KUKA KRL program: MyProgram_316().src

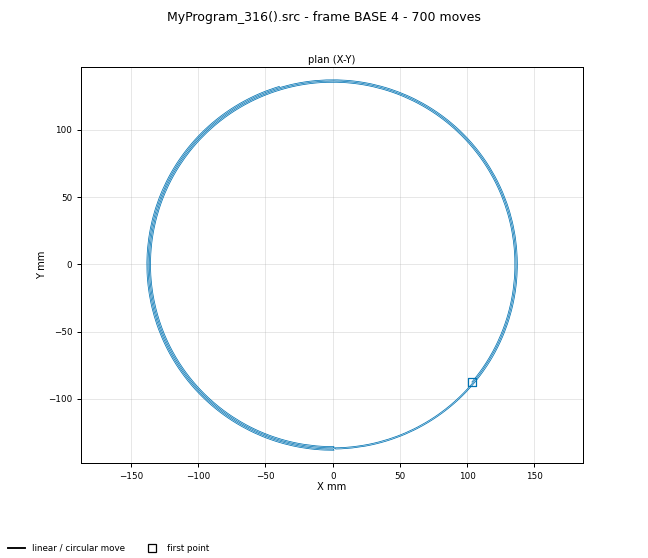
[picture p0: tool path of MyProgram_316().src in frame BASE 4, 700 of 700 moves have a stored position in this frame; points joined in program order, loops and branches not executed]
&ACCESS RVP
&REL 1
&PARAM TEMPLATE = C:\KRC\Roboter\Template\vorgabe
&PARAM EDITMASK = *
DEF MyProgram_316()
; ---- Setting reference (Base) ----
$BASE = BASE_DATA[4]

; --------------------------
; ---- Setting tool (TCP) ----
$TOOL = TOOL_DATA[3]
; --------------------------

$VEL.CP = VEL_APROX_PRINT
Startdeposition()
$VEL.CP = VEL_PRINT
LIN {X 103.5181,Y -87.4443,Z 184,A -35.435,B 3.7699,C 0.2794,E1 3.9046,E2 488.1643} C_DIS
LIN {X 106.5968,Y -83.6627,Z 184,A -33.5084,B 3.7701,C 0.2762,E1 3.9079,E2 486.2534} C_DIS
LIN {X 109.2391,Y -80.182,Z 184,A -31.7632,B 3.7704,C 0.2731,E1 3.9108,E2 484.52} C_DIS
LIN {X 111.321,Y -77.2656,Z 184,A -29.7761,B 3.771,C 0.2642,E1 3.9141,E2 482.4703} C_DIS
LIN {X 113.9076,Y -73.3999,Z 184,A -28.2787,B 3.771,C 0.2647,E1 3.9163,E2 481.0323} C_DIS
LIN {X 116.3066,Y -69.5351,Z 184,A -26.5939,B 3.7711,C 0.2627,E1 3.9187,E2 479.3768} C_DIS
LIN {X 119.2726,Y -64.315,Z 184,A -23.9196,B 3.7716,C 0.2548,E1 3.9223,E2 476.683} C_DIS
LIN {X 121.3738,Y -60.2518,Z 184,A -22.1723,B 3.7718,C 0.2519,E1 3.9245,E2 474.9581} C_DIS
LIN {X 122.8506,Y -57.1807,Z 184,A -20.8286,B 3.772,C 0.2493,E1 3.9261,E2 473.6257} C_DIS
LIN {X 124.2779,Y -54.0078,Z 184,A -19.6123,B 3.772,C 0.2483,E1 3.9274,E2 472.4408} C_DIS
LIN {X 125.1592,Y -51.9333,Z 184,A -18.3421,B 3.7725,C 0.2422,E1 3.9288,E2 471.1292} C_DIS
LIN {X 126.782,Y -47.8354,Z 184,A -16.8653,B 3.7725,C 0.2417,E1 3.9303,E2 469.7006} C_DIS
LIN {X 128.1212,Y -44.1231,Z 184,A -14.9406,B 3.773,C 0.2343,E1 3.9321,E2 467.7417} C_DIS
LIN {X 129.4777,Y -39.9682,Z 184,A -13.2527,B 3.7732,C 0.2311,E1 3.9335,E2 466.0729} C_DIS
LIN {X 130.4392,Y -36.7082,Z 184,A -11.883,B 3.7734,C 0.2279,E1 3.9346,E2 464.7107} C_DIS
LIN {X 131.3258,Y -33.3972,Z 184,A -10.4346,B 3.7736,C 0.2239,E1 3.9356,E2 463.2613} C_DIS
LIN {X 132.2992,Y -29.3141,Z 184,A -8.6511,B 3.7739,C 0.2189,E1 3.9367,E2 461.4754} C_DIS
LIN {X 133.0621,Y -25.6197,Z 184,A -7.2855,B 3.7739,C 0.2171,E1 3.9374,E2 460.1378} C_DIS
LIN {X 133.6399,Y -22.4114,Z 184,A -5.8945,B 3.7742,C 0.2131,E1 3.9381,E2 458.7442} C_DIS
LIN {X 134.2034,Y -18.7486,Z 184,A -4.3975,B 3.7744,C 0.2095,E1 3.9387,E2 457.2549} C_DIS
LIN {X 135.083,Y -10.7221,Z 184,A -1.0365,B 3.7749,C 0.2006,E1 3.9397,E2 453.8983} C_DIS
LIN {X 135.3222,Y -7.0634,Z 184,A 0.376,B 3.7751,C 0.1977,E1 3.9399,E2 452.5023} C_DIS
LIN {X 135.4633,Y -3.4258,Z 184,A 2.0383,B 3.7754,C 0.192,E1 3.94,E2 450.8232} C_DIS
LIN {X 135.4418,Y 4.2013,Z 184,A 5.0751,B 3.7757,C 0.185,E1 3.94,E2 447.8082} C_DIS
LIN {X 135.3131,Y 7.2441,Z 184,A 6.7756,B 3.7761,C 0.1767,E1 3.9397,E2 446.0544} C_DIS
LIN {X 134.9595,Y 12.1833,Z 184,A 8.2582,B 3.7761,C 0.1778,E1 3.9393,E2 444.6481} C_DIS
LIN {X 134.3821,Y 17.4175,Z 184,A 10.3473,B 3.7763,C 0.1731,E1 3.9386,E2 442.5749} C_DIS
LIN {X 133.9505,Y 20.4746,Z 184,A 11.6618,B 3.7764,C 0.1693,E1 3.9381,E2 441.2585} C_DIS
LIN {X 133.4035,Y 23.778,Z 184,A 12.9257,B 3.7765,C 0.1671,E1 3.9375,E2 440.0129} C_DIS
LIN {X 132.7476,Y 27.2026,Z 184,A 14.4382,B 3.7767,C 0.1626,E1 3.9367,E2 438.4947} C_DIS
LIN {X 131.8443,Y 31.2913,Z 184,A 16.18,B 3.7769,C 0.158,E1 3.9356,E2 436.7555} C_DIS
LIN {X 130.9715,Y 34.7611,Z 184,A 17.5774,B 3.777,C 0.1552,E1 3.9346,E2 435.3717} C_DIS
LIN {X 130.0827,Y 37.9517,Z 184,A 18.9487,B 3.7772,C 0.1517,E1 3.9336,E2 434.0034} C_DIS
LIN {X 129.068,Y 41.2706,Z 184,A 20.3738,B 3.7773,C 0.1482,E1 3.9324,E2 432.5828} C_DIS
LIN {X 128.1625,Y 44.0039,Z 184,A 21.9177,B 3.7776,C 0.1413,E1 3.931,E2 430.9974} C_DIS
LIN {X 126.8571,Y 47.635,Z 184,A 23.0833,B 3.7776,C 0.1422,E1 3.9299,E2 429.8894} C_DIS
LIN {X 125.7062,Y 50.594,Z 184,A 24.4415,B 3.7776,C 0.1384,E1 3.9285,E2 428.5286} C_DIS
LIN {X 124.1044,Y 54.4093,Z 184,A 26.2365,B 3.7779,C 0.1334,E1 3.9265,E2 426.7272} C_DIS
LIN {X 122.8136,Y 57.2608,Z 184,A 27.4747,B 3.7779,C 0.1309,E1 3.9251,E2 425.4991} C_DIS
LIN {X 121.1492,Y 60.7072,Z 184,A 29.0707,B 3.7781,C 0.1271,E1 3.9231,E2 423.9053} C_DIS
LIN {X 119.1914,Y 64.4661,Z 184,A 30.7766,B 3.7782,C 0.1235,E1 3.9208,E2 422.2093} C_DIS
LIN {X 116.2038,Y 69.7076,Z 184,A 33.2579,B 3.7784,C 0.118,E1 3.9174,E2 419.7358} C_DIS
LIN {X 113.8832,Y 73.4375,Z 184,A 34.9973,B 3.7784,C 0.1148,E1 3.9148,E2 418.0104} C_DIS
LIN {X 112.1478,Y 76.0606,Z 184,A 36.3024,B 3.7786,C 0.1119,E1 3.9128,E2 416.708} C_DIS
LIN {X 109.5386,Y 79.7729,Z 184,A 38.1589,B 3.7786,C 0.1081,E1 3.9098,E2 414.8587} C_DIS
LIN {X 106.995,Y 83.153,Z 184,A 39.8979,B 3.7788,C 0.1046,E1 3.9068,E2 413.1252} C_DIS
LIN {X 104.2275,Y 86.5968,Z 184,A 41.7072,B 3.7788,C 0.1011,E1 3.9036,E2 411.3227} C_DIS
LIN {X 101.3001,Y 90.004,Z 184,A 43.5795,B 3.779,C 0.0973,E1 3.9002,E2 409.4534} C_DIS
LIN {X 98.7892,Y 92.753,Z 184,A 45.5297,B 3.7792,C 0.09,E1 3.8964,E2 407.4564} C_DIS
LIN {X 95.608,Y 96.0284,Z 184,A 46.8132,B 3.7791,C 0.0928,E1 3.894,E2 406.2524} C_DIS
LIN {X 90.6851,Y 100.691,Z 184,A 49.8084,B 3.7793,C 0.0858,E1 3.8879,E2 403.2412} C_DIS
LIN {X 87.3464,Y 103.6004,Z 184,A 51.6137,B 3.7793,C 0.083,E1 3.884,E2 401.4439} C_DIS
LIN {X 84.0447,Y 106.2967,Z 184,A 53.3461,B 3.7793,C 0.0804,E1 3.8803,E2 399.72} C_DIS
LIN {X 80.6714,Y 108.8786,Z 184,A 55.1005,B 3.7794,C 0.0777,E1 3.8764,E2 397.9706} C_DIS
LIN {X 77.034,Y 111.4822,Z 184,A 56.9839,B 3.7794,C 0.0746,E1 3.8721,E2 396.0881} C_DIS
LIN {X 73.3256,Y 113.9552,Z 184,A 58.8067,B 3.7795,C 0.0722,E1 3.8678,E2 394.2729} C_DIS
LIN {X 69.7051,Y 116.2053,Z 184,A 60.6036,B 3.7795,C 0.0695,E1 3.8635,E2 392.4767} C_DIS
LIN {X 66.7818,Y 117.9097,Z 184,A 61.9456,B 3.7796,C 0.0682,E1 3.8603,E2 391.1456} C_DIS
LIN {X 63.2705,Y 119.8278,Z 184,A 63.5525,B 3.7796,C 0.0667,E1 3.8564,E2 389.549} C_DIS
LIN {X 60.3352,Y 121.3327,Z 184,A 64.9003,B 3.7796,C 0.0652,E1 3.853,E2 388.2071} C_DIS
LIN {X 57.0324,Y 122.9191,Z 184,A 66.4113,B 3.7796,C 0.0636,E1 3.8492,E2 386.7009} C_DIS
LIN {X 54.1496,Y 124.2167,Z 184,A 67.7281,B 3.7797,C 0.0622,E1 3.8459,E2 385.3867} C_DIS
LIN {X 50.7905,Y 125.627,Z 184,A 69.2033,B 3.7797,C 0.061,E1 3.8421,E2 383.9196} C_DIS
LIN {X 47.6823,Y 126.8394,Z 184,A 70.6206,B 3.7797,C 0.0594,E1 3.8384,E2 382.5017} C_DIS
LIN {X 44.4026,Y 128.0243,Z 184,A 72.1122,B 3.7797,C 0.0578,E1 3.8344,E2 381.0083} C_DIS
LIN {X 41.1802,Y 129.0969,Z 184,A 73.6768,B 3.7798,C 0.0552,E1 3.8302,E2 379.4284} C_DIS
LIN {X 37.2623,Y 130.2842,Z 184,A 75.3555,B 3.7798,C 0.0542,E1 3.8258,E2 377.7565} C_DIS
LIN {X 33.5935,Y 131.276,Z 184,A 76.8272,B 3.7798,C 0.0542,E1 3.8218,E2 376.3015} C_DIS
LIN {X 30.4525,Y 132.0401,Z 184,A 78.1762,B 3.7798,C 0.0533,E1 3.8182,E2 374.9551} C_DIS
LIN {X 26.9784,Y 132.7932,Z 184,A 79.7173,B 3.7798,C 0.0519,E1 3.8139,E2 373.4097} C_DIS
LIN {X 22.9319,Y 133.553,Z 184,A 81.4911,B 3.7798,C 0.0506,E1 3.809,E2 371.6326} C_DIS
LIN {X 19.2145,Y 134.1368,Z 184,A 83.0044,B 3.7798,C 0.0505,E1 3.8049,E2 370.1291} C_DIS
LIN {X 15.1542,Y 134.6577,Z 184,A 85.3116,B 3.78,C 0.0449,E1 3.7983,E2 367.7527} C_DIS
LIN {X 10.2568,Y 135.118,Z 184,A 86.7787,B 3.78,C 0.0494,E1 3.7944,E2 366.3607} C_DIS
LIN {X 6.746,Y 135.3382,Z 184,A 88.2689,B 3.78,C 0.049,E1 3.7903,E2 364.8707} C_DIS
LIN {X 2.8347,Y 135.4778,Z 184,A 90.1909,B 3.78,C 0.0465,E1 3.7848,E2 362.9171} C_DIS
LIN {X -4.5052,Y 135.4333,Z 184,A 93.1017,B 3.78,C 0.0479,E1 3.7767,E2 360.0311} C_DIS
LIN {X -8.3822,Y 135.2467,Z 184,A 94.6551,B 3.78,C 0.0487,E1 3.7724,E2 358.489} C_DIS
LIN {X -11.9873,Y 134.9761,Z 184,A 96.6447,B 3.78,C 0.0454,E1 3.7667,E2 356.4445} C_DIS
LIN {X -16.0503,Y 134.5522,Z 184,A 97.9717,B 3.78,C 0.0489,E1 3.7632,E2 355.1668} C_DIS
LIN {X -20.4686,Y 133.9514,Z 184,A 99.7685,B 3.7799,C 0.0501,E1 3.7583,E2 353.3815} C_DIS
LIN {X -23.5464,Y 133.4449,Z 184,A 101.1595,B 3.7799,C 0.0501,E1 3.7544,E2 351.9826} C_DIS
LIN {X -26.9594,Y 132.797,Z 184,A 102.6559,B 3.7799,C 0.0506,E1 3.7503,E2 350.4837} C_DIS
LIN {X -30.9686,Y 131.9221,Z 184,A 104.4857,B 3.7799,C 0.0508,E1 3.7453,E2 348.6435} C_DIS
LIN {X -34.5894,Y 131.0173,Z 184,A 105.9655,B 3.7799,C 0.0525,E1 3.7413,E2 347.1765} C_DIS
LIN {X -37.9806,Y 130.0742,Z 184,A 107.5309,B 3.7799,C 0.053,E1 3.7371,E2 345.6026} C_DIS
LIN {X -42.695,Y 128.6039,Z 184,A 109.5217,B 3.7799,C 0.0553,E1 3.7318,E2 343.6248} C_DIS
LIN {X -45.7334,Y 127.5552,Z 184,A 111.6211,B 3.7799,C 0.0513,E1 3.7261,E2 341.4366} C_DIS
LIN {X -50.6638,Y 125.6781,Z 184,A 113.2742,B 3.7798,C 0.0575,E1 3.722,E2 339.8551} C_DIS
LIN {X -54.6362,Y 124.005,Z 184,A 115.1537,B 3.7798,C 0.059,E1 3.7171,E2 337.97} C_DIS
LIN {X -57.8691,Y 122.5288,Z 184,A 116.6209,B 3.7798,C 0.0609,E1 3.7134,E2 336.508} C_DIS
LIN {X -61.0853,Y 120.9568,Z 184,A 118.6584,B 3.7798,C 0.0592,E1 3.7082,E2 334.4081} C_DIS
LIN {X -65.2213,Y 118.7799,Z 184,A 120.237,B 3.7797,C 0.0644,E1 3.7044,E2 332.8792} C_DIS
LIN {X -69.0275,Y 116.6091,Z 184,A 122.1205,B 3.7797,C 0.0667,E1 3.6999,E2 330.9933} C_DIS
LIN {X -73.0206,Y 114.1504,Z 184,A 124.4662,B 3.7797,C 0.0673,E1 3.6942,E2 328.6049} C_DIS
LIN {X -76.3633,Y 111.9425,Z 184,A 125.8969,B 3.7796,C 0.0715,E1 3.691,E2 327.2075} C_DIS
LIN {X -79.8005,Y 109.5186,Z 184,A 128.3863,B 3.7796,C 0.0699,E1 3.6852,E2 324.6327} C_DIS
LIN {X -84.4566,Y 105.9683,Z 184,A 130.1256,B 3.7794,C 0.0787,E1 3.6816,E2 322.9852} C_DIS
LIN {X -87.6625,Y 103.3326,Z 184,A 132.0123,B 3.7794,C 0.081,E1 3.6775,E2 321.0838} C_DIS
LIN {X -91.0944,Y 100.3202,Z 184,A 133.9814,B 3.7793,C 0.0843,E1 3.6734,E2 319.1115} C_DIS
LIN {X -93.5494,Y 98.0349,Z 184,A 135.4341,B 3.7793,C 0.0868,E1 3.6704,E2 317.6557} C_DIS
LIN {X -98.0838,Y 93.4983,Z 184,A 138.206,B 3.7791,C 0.0918,E1 3.665,E2 314.8787} C_DIS
LIN {X -100.7109,Y 90.6629,Z 184,A 140.4369,B 3.7791,C 0.0918,E1 3.6607,E2 312.5761} C_DIS
LIN {X -103.9243,Y 86.9603,Z 184,A 142.3254,B 3.779,C 0.0972,E1 3.6573,E2 310.7119} C_DIS
LIN {X -106.2486,Y 84.1053,Z 184,A 143.8562,B 3.7789,C 0.1007,E1 3.6547,E2 309.1855} C_DIS
LIN {X -108.2291,Y 81.5401,Z 184,A 145.0338,B 3.7788,C 0.1049,E1 3.6527,E2 308.0327} C_DIS
LIN {X -109.8686,Y 79.3177,Z 184,A 146.4136,B 3.7788,C 0.1063,E1 3.6504,E2 306.6279} C_DIS
LIN {X -113.4809,Y 74.0572,Z 184,A 149.1427,B 3.7786,C 0.1124,E1 3.6462,E2 303.8971} C_DIS
LIN {X -116.0885,Y 69.8989,Z 184,A 151.1973,B 3.7784,C 0.1175,E1 3.6432,E2 301.8467} C_DIS
LIN {X -118.3289,Y 66.0361,Z 184,A 153.1725,B 3.7783,C 0.1217,E1 3.6404,E2 299.8623} C_DIS
LIN {X -120.4533,Y 62.0743,Z 184,A 155.1282,B 3.7781,C 0.1261,E1 3.6379,E2 297.9014} C_DIS
LIN {X -122.1757,Y 58.6082,Z 184,A 156.6266,B 3.778,C 0.131,E1 3.6361,E2 296.4212} C_DIS
LIN {X -124.6543,Y 53.1374,Z 184,A 159.4282,B 3.7778,C 0.1361,E1 3.6329,E2 293.5895} C_DIS
LIN {X -126.1375,Y 49.5109,Z 184,A 161.1089,B 3.7776,C 0.1403,E1 3.6311,E2 291.9072} C_DIS
LIN {X -127.6232,Y 45.5447,Z 184,A 163.4121,B 3.7776,C 0.1424,E1 3.6289,E2 289.5419} C_DIS
LIN {X -128.9736,Y 41.5661,Z 184,A 164.6478,B 3.7773,C 0.15,E1 3.6279,E2 288.3746} C_DIS
LIN {X -130.6703,Y 35.8819,Z 184,A 167.4986,B 3.7771,C 0.155,E1 3.6256,E2 285.4835} C_DIS
LIN {X -131.6553,Y 32.0754,Z 184,A 169.697,B 3.777,C 0.1568,E1 3.6241,E2 283.2197} C_DIS
LIN {X -132.7065,Y 27.4043,Z 184,A 171.0506,B 3.7766,C 0.1659,E1 3.6234,E2 281.9511} C_DIS
LIN {X -133.4038,Y 23.7763,Z 184,A 172.8553,B 3.7765,C 0.169,E1 3.6224,E2 280.1176} C_DIS
LIN {X -134.0865,Y 19.5668,Z 184,A 174.7057,B 3.7762,C 0.1738,E1 3.6216,E2 278.2626} C_DIS
LIN {X -134.5631,Y 15.9588,Z 184,A 176.3185,B 3.7761,C 0.1777,E1 3.6211,E2 276.6417} C_DIS
LIN {X -134.9882,Y 11.8438,Z 184,A 178.1693,B 3.7758,C 0.1821,E1 3.6206,E2 274.7795} C_DIS
LIN {X -135.2793,Y 7.8531,Z 184,A 179.9378,B 3.7756,C 0.1865,E1 3.6202,E2 273.0026} C_DIS
LIN {X -135.4525,Y 3.8144,Z 184,A -178.3293,B 3.7754,C 0.1912,E1 3.6201,E2 271.268} C_DIS
LIN {X -135.5061,Y -0.3615,Z 184,A -176.5359,B 3.7751,C 0.1961,E1 3.6201,E2 269.4723} C_DIS
LIN {X -135.4553,Y -3.7156,Z 184,A -175.0132,B 3.775,C 0.1996,E1 3.6201,E2 267.9375} C_DIS
LIN {X -135.2704,Y -7.9973,Z 184,A -173.16,B 3.7747,C 0.2045,E1 3.6204,E2 266.0804} C_DIS
LIN {X -135.0247,Y -11.4122,Z 184,A -171.6847,B 3.7745,C 0.2084,E1 3.6207,E2 264.6025} C_DIS
LIN {X -134.675,Y -14.9935,Z 184,A -169.9572,B 3.7743,C 0.2116,E1 3.6212,E2 262.8501} C_DIS
LIN {X -134.1557,Y -19.0822,Z 184,A -168.2428,B 3.774,C 0.2166,E1 3.6219,E2 261.1403} C_DIS
LIN {X -133.607,Y -22.6086,Z 184,A -166.6738,B 3.7738,C 0.2205,E1 3.6226,E2 259.5647} C_DIS
LIN {X -132.8478,Y -26.7098,Z 184,A -164.7999,B 3.7735,C 0.2248,E1 3.6236,E2 257.6778} C_DIS
LIN {X -132.0995,Y -30.1923,Z 184,A -163.2973,B 3.7733,C 0.2289,E1 3.6245,E2 256.1766} C_DIS
LIN {X -131.4851,Y -32.7696,Z 184,A -161.5672,B 3.7733,C 0.2288,E1 3.6257,E2 254.3697} C_DIS
LIN {X -130.2917,Y -37.2355,Z 184,A -160.0518,B 3.7728,C 0.2364,E1 3.6268,E2 252.9113} C_DIS
LIN {X -128.7739,Y -42.1845,Z 184,A -157.8959,B 3.7725,C 0.2424,E1 3.6286,E2 250.7607} C_DIS
LIN {X -127.0289,Y -47.1764,Z 184,A -155.4027,B 3.7722,C 0.2469,E1 3.631,E2 248.236} C_DIS
LIN {X -125.6609,Y -50.7063,Z 184,A -153.8514,B 3.7719,C 0.2514,E1 3.6326,E2 246.6917} C_DIS
LIN {X -124.315,Y -53.9222,Z 184,A -152.2845,B 3.7717,C 0.2546,E1 3.6343,E2 245.1137} C_DIS
LIN {X -122.6707,Y -57.5696,Z 184,A -150.4266,B 3.7714,C 0.258,E1 3.6365,E2 243.2354} C_DIS
LIN {X -120.9111,Y -61.175,Z 184,A -149.0155,B 3.771,C 0.2638,E1 3.6382,E2 241.8613} C_DIS
LIN {X -119.1588,Y -64.5265,Z 184,A -147.2309,B 3.7708,C 0.2667,E1 3.6406,E2 240.0538} C_DIS
LIN {X -116.6686,Y -68.9266,Z 184,A -144.8564,B 3.7706,C 0.2705,E1 3.6439,E2 237.6498} C_DIS
LIN {X -114.3702,Y -72.6771,Z 184,A -142.8945,B 3.7703,C 0.2742,E1 3.6468,E2 235.6755} C_DIS
LIN {X -111.9924,Y -76.2901,Z 184,A -141.0164,B 3.77,C 0.2781,E1 3.6498,E2 233.7916} C_DIS
LIN {X -109.5736,Y -79.7246,Z 184,A -139.2203,B 3.7697,C 0.282,E1 3.6527,E2 231.9934} C_DIS
LIN {X -106.9244,Y -83.2441,Z 184,A -137.2892,B 3.7694,C 0.2856,E1 3.656,E2 230.0541} C_DIS
LIN {X -104.1668,Y -86.67,Z 184,A -135.383,B 3.7692,C 0.2893,E1 3.6594,E2 228.1423} C_DIS
LIN {X -101.1471,Y -90.1759,Z 184,A -133.0311,B 3.769,C 0.2908,E1 3.6638,E2 225.7397} C_DIS
LIN {X -98.49,Y -93.0702,Z 184,A -131.7079,B 3.7686,C 0.2963,E1 3.6663,E2 224.4605} C_DIS
LIN {X -95.4751,Y -96.1604,Z 184,A -129.7354,B 3.7684,C 0.2988,E1 3.6702,E2 222.4694} C_DIS
LIN {X -92.0118,Y -99.4802,Z 184,A -127.6647,B 3.7681,C 0.3023,E1 3.6744,E2 220.3935} C_DIS
LIN {X -88.6199,Y -102.5129,Z 184,A -125.7108,B 3.7679,C 0.3055,E1 3.6785,E2 218.4359} C_DIS
LIN {X -85.1174,Y -105.4389,Z 184,A -123.758,B 3.7676,C 0.3086,E1 3.6827,E2 216.4802} C_DIS
LIN {X -81.5764,Y -108.2018,Z 184,A -121.8385,B 3.7674,C 0.3116,E1 3.687,E2 214.5582} C_DIS
LIN {X -77.8987,Y -110.8791,Z 184,A -119.8504,B 3.7672,C 0.3141,E1 3.6915,E2 212.5617} C_DIS
LIN {X -74.2217,Y -113.3736,Z 184,A -117.9263,B 3.767,C 0.3165,E1 3.696,E2 210.6318} C_DIS
LIN {X -70.3633,Y -115.8077,Z 184,A -116.207,B 3.7666,C 0.3206,E1 3.7,E2 208.9396} C_DIS
LIN {X -68.2455,Y -117.0683,Z 184,A -114.8236,B 3.7667,C 0.3196,E1 3.7035,E2 207.5118} C_DIS
LIN {X -63.8415,Y -119.527,Z 184,A -112.7187,B 3.7665,C 0.3224,E1 3.7086,E2 205.4103} C_DIS
LIN {X -60.7072,Y -121.1492,Z 184,A -111.2132,B 3.7663,C 0.324,E1 3.7124,E2 203.903} C_DIS
LIN {X -57.1333,Y -122.8725,Z 184,A -109.6227,B 3.7661,C 0.3265,E1 3.7164,E2 202.3236} C_DIS
LIN {X -54.0661,Y -124.2527,Z 184,A -108.2245,B 3.766,C 0.3281,E1 3.7199,E2 200.9283} C_DIS
LIN {X -50.9259,Y -125.5724,Z 184,A -106.6428,B 3.766,C 0.3284,E1 3.7241,E2 199.3279} C_DIS
LIN {X -46.873,Y -127.1425,Z 184,A -104.7358,B 3.7659,C 0.3295,E1 3.7291,E2 197.4116} C_DIS
LIN {X -43.7249,Y -128.2592,Z 184,A -103.2221,B 3.7659,C 0.3298,E1 3.7331,E2 195.8843} C_DIS
LIN {X -38.766,Y -129.8443,Z 184,A -101.0934,B 3.7657,C 0.3319,E1 3.7388,E2 193.7645} C_DIS
LIN {X -35.1377,Y -130.8711,Z 184,A -99.6095,B 3.7655,C 0.3337,E1 3.7427,E2 192.2947} C_DIS
LIN {X -31.8602,Y -131.7072,Z 184,A -98.2135,B 3.7654,C 0.3348,E1 3.7465,E2 190.9028} C_DIS
LIN {X -28.4852,Y -132.4782,Z 184,A -96.6735,B 3.7654,C 0.3348,E1 3.7508,E2 189.3523} C_DIS
LIN {X -24.5153,Y -133.2715,Z 184,A -94.8789,B 3.7654,C 0.3348,E1 3.7557,E2 187.5463} C_DIS
LIN {X -21.0207,Y -133.8659,Z 184,A -93.4272,B 3.7654,C 0.3357,E1 3.7597,E2 186.1002} C_DIS
LIN {X -12.4525,Y -134.9336,Z 184,A -89.6934,B 3.7654,C 0.3357,E1 3.7701,E2 182.3543} C_DIS
LIN {X -8.3999,Y -135.2456,Z 184,A -87.8487,B 3.7654,C 0.3347,E1 3.7753,E2 180.4924} C_DIS
LIN {X -3.6225,Y -135.4579,Z 184,A -85.4259,B 3.7657,C 0.331,E1 3.7822,E2 178.0158} C_DIS
LIN {X 0.9601,Y -135.4941,Z 184,A -85.2023,B 3.7644,C 0.3457,E1 3.7822,E2 178.0149} C_DIS
Enddeposition()
LIN {X 0.9601,Y -135.4941,Z 184,A -85.2026,B 3.7644,C 0.3457,E1 3.7822,E2 178.0154} C_DIS
Startdeposition()
$VEL.CP = VEL_PRINT
LIN {X 0.3837,Y -136.4071,Z 184,A -85.6049,B 3.698,C 0.3472,E1 3.7149,E2 178.4898} C_DIS
LIN {X -4.9994,Y -136.3158,Z 184,A -86.9807,B 3.6987,C 0.3398,E1 3.7113,E2 179.7514} C_DIS
LIN {X -11.1783,Y -135.9485,Z 184,A -89.729,B 3.6985,C 0.341,E1 3.7036,E2 182.5204} C_DIS
LIN {X -19.1236,Y -135.0598,Z 184,A -93.176,B 3.6985,C 0.3411,E1 3.694,E2 185.9804} C_DIS
LIN {X -22.669,Y -134.5102,Z 184,A -94.6664,B 3.6985,C 0.3405,E1 3.6898,E2 187.4692} C_DIS
LIN {X -26.3798,Y -133.834,Z 184,A -96.369,B 3.6985,C 0.3409,E1 3.6851,E2 189.1879} C_DIS
LIN {X -30.3642,Y -132.9843,Z 184,A -97.9709,B 3.6987,C 0.3392,E1 3.6808,E2 190.7759} C_DIS
LIN {X -33.567,Y -132.2121,Z 184,A -99.3949,B 3.6987,C 0.3388,E1 3.6769,E2 192.2056} C_DIS
LIN {X -37.1107,Y -131.2621,Z 184,A -100.8943,B 3.6989,C 0.3375,E1 3.6729,E2 193.7} C_DIS
LIN {X -40.2491,Y -130.3338,Z 184,A -102.5183,B 3.6988,C 0.3385,E1 3.6685,E2 195.3568} C_DIS
LIN {X -43.6729,Y -129.2278,Z 184,A -103.8767,B 3.699,C 0.3362,E1 3.6649,E2 196.6957} C_DIS
LIN {X -47.7093,Y -127.7912,Z 184,A -105.7782,B 3.699,C 0.3355,E1 3.6599,E2 198.6108} C_DIS
LIN {X -51.4947,Y -126.3144,Z 184,A -107.3588,B 3.6993,C 0.333,E1 3.6558,E2 200.1753} C_DIS
LIN {X -54.3414,Y -125.1152,Z 184,A -108.7378,B 3.6993,C 0.3323,E1 3.6522,E2 201.5651} C_DIS
LIN {X -57.5376,Y -123.678,Z 184,A -110.1947,B 3.6995,C 0.3307,E1 3.6485,E2 203.0203} C_DIS
LIN {X -60.5923,Y -122.2104,Z 184,A -111.6452,B 3.6996,C 0.3293,E1 3.6449,E2 204.4744} C_DIS
LIN {X -63.5016,Y -120.724,Z 184,A -113.0081,B 3.6998,C 0.3276,E1 3.6415,E2 205.8363} C_DIS
LIN {X -67.1135,Y -118.7568,Z 184,A -115.0141,B 3.6998,C 0.3274,E1 3.6365,E2 207.8785} C_DIS
LIN {X -71.5353,Y -116.1466,Z 184,A -117.1034,B 3.7001,C 0.324,E1 3.6315,E2 209.9592} C_DIS
LIN {X -75.29,Y -113.7489,Z 184,A -118.9736,B 3.7003,C 0.3214,E1 3.6272,E2 211.8293} C_DIS
LIN {X -78.7577,Y -111.3756,Z 184,A -120.7895,B 3.7005,C 0.319,E1 3.623,E2 213.6517} C_DIS
LIN {X -82.3707,Y -108.7309,Z 184,A -122.7201,B 3.7007,C 0.3164,E1 3.6186,E2 215.5887} C_DIS
LIN {X -85.9435,Y -105.9299,Z 184,A -124.6448,B 3.701,C 0.3133,E1 3.6144,E2 217.5156} C_DIS
LIN {X -89.3065,Y -103.1105,Z 184,A -126.5468,B 3.7012,C 0.3105,E1 3.6104,E2 219.425} C_DIS
LIN {X -92.623,Y -100.142,Z 184,A -128.4949,B 3.7015,C 0.3076,E1 3.6063,E2 221.383} C_DIS
LIN {X -95.912,Y -96.996,Z 184,A -130.3054,B 3.7018,C 0.3034,E1 3.6027,E2 223.1801} C_DIS
LIN {X -98.3561,Y -94.5172,Z 184,A -132.1449,B 3.7018,C 0.3029,E1 3.599,E2 225.068} C_DIS
LIN {X -100.5691,Y -92.1585,Z 184,A -133.3543,B 3.7021,C 0.2993,E1 3.5968,E2 226.258} C_DIS
LIN {X -103.1416,Y -89.2704,Z 184,A -135.0444,B 3.7024,C 0.2963,E1 3.5937,E2 227.9562} C_DIS
LIN {X -105.9965,Y -85.8609,Z 184,A -136.9694,B 3.7027,C 0.2927,E1 3.5902,E2 229.8879} C_DIS
LIN {X -108.8136,Y -82.2611,Z 184,A -138.9029,B 3.703,C 0.2886,E1 3.5869,E2 231.8227} C_DIS
LIN {X -111.2881,Y -78.8819,Z 184,A -140.7562,B 3.7033,C 0.2853,E1 3.5839,E2 233.6875} C_DIS
LIN {X -113.855,Y -75.1288,Z 184,A -142.6914,B 3.7036,C 0.281,E1 3.5809,E2 235.6253} C_DIS
LIN {X -116.2164,Y -71.4216,Z 184,A -144.5927,B 3.7039,C 0.277,E1 3.578,E2 237.5331} C_DIS
LIN {X -119.0092,Y -66.6643,Z 184,A -147.0142,B 3.7042,C 0.272,E1 3.5746,E2 239.967} C_DIS
LIN {X -121.2787,Y -62.4387,Z 184,A -148.9041,B 3.7047,C 0.2664,E1 3.5722,E2 241.8402} C_DIS
LIN {X -123.1322,Y -58.6959,Z 184,A -150.8616,B 3.7049,C 0.2631,E1 3.5698,E2 243.8228} C_DIS
LIN {X -124.5933,Y -55.5274,Z 184,A -152.3207,B 3.7052,C 0.2594,E1 3.5681,E2 245.2804} C_DIS
LIN {X -126.0051,Y -52.2453,Z 184,A -153.8959,B 3.7054,C 0.2559,E1 3.5664,E2 246.8644} C_DIS
LIN {X -127.3748,Y -48.8144,Z 184,A -155.8601,B 3.7055,C 0.254,E1 3.5643,E2 248.8801} C_DIS
LIN {X -128.6113,Y -45.4562,Z 184,A -157.2953,B 3.7058,C 0.2497,E1 3.563,E2 250.306} C_DIS
LIN {X -130.1808,Y -40.7477,Z 184,A -159.3693,B 3.7062,C 0.2441,E1 3.5612,E2 252.3776} C_DIS
LIN {X -131.4099,Y -36.5821,Z 184,A -161.4985,B 3.7064,C 0.2408,E1 3.5596,E2 254.5441} C_DIS
LIN {X -132.3787,Y -32.9109,Z 184,A -162.8408,B 3.7068,C 0.2351,E1 3.5587,E2 255.8538} C_DIS
LIN {X -133.2756,Y -29.0603,Z 184,A -164.5238,B 3.707,C 0.2307,E1 3.5576,E2 257.5387} C_DIS
LIN {X -134.0075,Y -25.472,Z 184,A -166.1504,B 3.7073,C 0.2269,E1 3.5567,E2 259.1754} C_DIS
LIN {X -134.7597,Y -21.1357,Z 184,A -168.0657,B 3.7076,C 0.2221,E1 3.5559,E2 261.0981} C_DIS
LIN {X -135.3,Y -17.3464,Z 184,A -169.6828,B 3.7078,C 0.2176,E1 3.5553,E2 262.7153} C_DIS
LIN {X -135.7574,Y -13.2984,Z 184,A -171.4955,B 3.7081,C 0.2134,E1 3.5547,E2 264.5396} C_DIS
LIN {X -136.052,Y -9.8344,Z 184,A -173.0048,B 3.7083,C 0.2095,E1 3.5544,E2 266.0542} C_DIS
LIN {X -136.2412,Y -6.7259,Z 184,A -174.342,B 3.7085,C 0.2059,E1 3.5542,E2 267.3941} C_DIS
LIN {X -136.3719,Y -3.1606,Z 184,A -176.0368,B 3.7087,C 0.2027,E1 3.554,E2 269.1125} C_DIS
LIN {X -136.4036,Y 1.007,Z 184,A -177.7269,B 3.709,C 0.1974,E1 3.554,E2 270.7938} C_DIS
LIN {X -136.3162,Y 4.9876,Z 184,A -179.5129,B 3.7092,C 0.1933,E1 3.5542,E2 272.5928} C_DIS
LIN {X -136.1363,Y 8.5914,Z 184,A 178.9992,B 3.7094,C 0.1889,E1 3.5544,E2 274.0762} C_DIS
LIN {X -135.8983,Y 11.7732,Z 184,A 177.6022,B 3.7096,C 0.1854,E1 3.5547,E2 275.4793} C_DIS
LIN {X -135.5827,Y 14.9779,Z 184,A 176.1472,B 3.7097,C 0.1821,E1 3.5551,E2 276.9461} C_DIS
LIN {X -135.104,Y 18.8145,Z 184,A 174.3912,B 3.7099,C 0.1782,E1 3.5558,E2 278.7173} C_DIS
LIN {X -134.5359,Y 22.5147,Z 184,A 172.8206,B 3.7101,C 0.1738,E1 3.5565,E2 280.2865} C_DIS
LIN {X -133.8763,Y 26.1584,Z 184,A 170.6056,B 3.7101,C 0.1727,E1 3.5577,E2 282.5815} C_DIS
LIN {X -132.8811,Y 30.8161,Z 184,A 169.2499,B 3.7106,C 0.164,E1 3.5585,E2 283.8564} C_DIS
LIN {X -132.2273,Y 33.5073,Z 184,A 167.9395,B 3.7106,C 0.1615,E1 3.5594,E2 285.1841} C_DIS
LIN {X -131.2526,Y 37.1446,Z 184,A 165.7846,B 3.7108,C 0.1601,E1 3.561,E2 287.4081} C_DIS
LIN {X -130.0458,Y 41.1701,Z 184,A 164.6348,B 3.7111,C 0.1523,E1 3.5619,E2 288.4811} C_DIS
LIN {X -129.1414,Y 43.9299,Z 184,A 162.8763,B 3.7111,C 0.1517,E1 3.5635,E2 290.3048} C_DIS
LIN {X -128.0635,Y 46.9796,Z 184,A 161.7804,B 3.7113,C 0.1468,E1 3.5646,E2 291.3676} C_DIS
LIN {X -127.0409,Y 49.6732,Z 184,A 160.4784,B 3.7114,C 0.1441,E1 3.5659,E2 292.6797} C_DIS
LIN {X -124.6593,Y 55.3798,Z 184,A 157.6421,B 3.7116,C 0.1385,E1 3.569,E2 295.5433} C_DIS
LIN {X -123.0145,Y 58.9421,Z 184,A 156.1044,B 3.7118,C 0.1338,E1 3.5708,E2 297.0662} C_DIS
LIN {X -121.5187,Y 61.9673,Z 184,A 154.6248,B 3.7119,C 0.1305,E1 3.5727,E2 298.5523} C_DIS
LIN {X -119.7672,Y 65.2925,Z 184,A 152.9119,B 3.712,C 0.1273,E1 3.575,E2 300.2803} C_DIS
LIN {X -117.4932,Y 69.3015,Z 184,A 150.899,B 3.7122,C 0.123,E1 3.5778,E2 302.301} C_DIS
LIN {X -115.1757,Y 73.0887,Z 184,A 148.5484,B 3.7122,C 0.1211,E1 3.5814,E2 304.709} C_DIS
LIN {X -112.7574,Y 76.767,Z 184,A 146.5583,B 3.7123,C 0.1176,E1 3.5845,E2 306.7146} C_DIS
LIN {X -109.997,Y 80.6718,Z 184,A 145.3746,B 3.7126,C 0.1086,E1 3.5863,E2 307.7968} C_DIS
LIN {X -104.2884,Y 87.9279,Z 184,A 140.7817,B 3.7128,C 0.1041,E1 3.5944,E2 312.4734} C_DIS
LIN {X -102.16,Y 90.3915,Z 184,A 139.9572,B 3.7129,C 0.0982,E1 3.5958,E2 313.2312} C_DIS
LIN {X -98.8015,Y 94.0512,Z 184,A 137.4639,B 3.7129,C 0.0963,E1 3.6006,E2 315.7722} C_DIS
LIN {X -94.5206,Y 98.3528,Z 184,A 134.7958,B 3.7131,C 0.092,E1 3.606,E2 318.4527} C_DIS
LIN {X -91.2527,Y 101.392,Z 184,A 132.9277,B 3.7131,C 0.0885,E1 3.6098,E2 320.3186} C_DIS
LIN {X -88.0072,Y 104.2219,Z 184,A 131.0511,B 3.7132,C 0.0856,E1 3.6138,E2 322.202} C_DIS
LIN {X -81.572,Y 109.3312,Z 184,A 127.681,B 3.7134,C 0.0793,E1 3.6212,E2 325.5598} C_DIS
LIN {X -78.6497,Y 111.4518,Z 184,A 125.9551,B 3.7134,C 0.0782,E1 3.6252,E2 327.3098} C_DIS
LIN {X -74.8059,Y 114.0676,Z 184,A 123.818,B 3.7134,C 0.0763,E1 3.6302,E2 329.4676} C_DIS
LIN {X -69.6193,Y 117.3052,Z 184,A 121.6029,B 3.7135,C 0.0705,E1 3.6353,E2 331.6384} C_DIS
LIN {X -67.1805,Y 118.7191,Z 184,A 119.9435,B 3.7135,C 0.0719,E1 3.6395,E2 333.3541} C_DIS
LIN {X -60.8434,Y 122.0865,Z 184,A 117.2757,B 3.7136,C 0.066,E1 3.646,E2 335.9782} C_DIS
LIN {X -58.4928,Y 123.2292,Z 184,A 116.0327,B 3.7136,C 0.0657,E1 3.6492,E2 337.2379} C_DIS
LIN {X -55.3961,Y 124.652,Z 184,A 114.5563,B 3.7136,C 0.0644,E1 3.6529,E2 338.7187} C_DIS
LIN {X -48.0379,Y 127.6682,Z 184,A 111.4529,B 3.7137,C 0.0596,E1 3.6609,E2 341.7917} C_DIS
LIN {X -45.7117,Y 128.5206,Z 184,A 110.1639,B 3.7137,C 0.0603,E1 3.6644,E2 343.1099} C_DIS
LIN {X -41.8883,Y 129.8164,Z 184,A 108.4343,B 3.7137,C 0.0592,E1 3.669,E2 344.8425} C_DIS
LIN {X -37.6851,Y 131.0994,Z 184,A 106.6314,B 3.7137,C 0.0575,E1 3.6738,E2 346.6391} C_DIS
LIN {X -33.2281,Y 132.2982,Z 184,A 104.6477,B 3.7137,C 0.0566,E1 3.6791,E2 348.6271} C_DIS
LIN {X -30.0152,Y 133.064,Z 184,A 103.276,B 3.7137,C 0.0558,E1 3.6829,E2 349.9961} C_DIS
LIN {X -27.1142,Y 133.6848,Z 184,A 101.9329,B 3.7137,C 0.0558,E1 3.6866,E2 351.3501} C_DIS
LIN {X -23.7555,Y 134.3226,Z 184,A 100.494,B 3.7137,C 0.0553,E1 3.6905,E2 352.7887} C_DIS
LIN {X -19.5528,Y 134.9985,Z 184,A 98.6675,B 3.7138,C 0.0549,E1 3.6956,E2 354.6188} C_DIS
LIN {X -15.8929,Y 135.4782,Z 184,A 96.6242,B 3.7138,C 0.0583,E1 3.7014,E2 356.7201} C_DIS
LIN {X -11.3232,Y 135.9363,Z 184,A 95.4244,B 3.7138,C 0.0524,E1 3.7045,E2 357.832} C_DIS
LIN {X -7.4163,Y 136.2064,Z 184,A 93.6949,B 3.7138,C 0.0529,E1 3.7094,E2 359.5708} C_DIS
LIN {X 1.0775,Y 136.4032,Z 184,A 90.0742,B 3.7138,C 0.0535,E1 3.7195,E2 363.1963} C_DIS
LIN {X 6.5396,Y 136.2505,Z 184,A 87.9346,B 3.7138,C 0.0527,E1 3.7254,E2 365.3163} C_DIS
LIN {X 13.0678,Y 135.7796,Z 184,A 84.8736,B 3.7138,C 0.056,E1 3.7341,E2 368.4137} C_DIS
LIN {X 16.9237,Y 135.355,Z 184,A 83.4125,B 3.7138,C 0.0553,E1 3.7381,E2 369.8542} C_DIS
LIN {X 21.067,Y 134.7704,Z 184,A 81.6314,B 3.7138,C 0.0564,E1 3.743,E2 371.6375} C_DIS
LIN {X 24.4241,Y 134.203,Z 184,A 80.2147,B 3.7138,C 0.0571,E1 3.7469,E2 373.0521} C_DIS
LIN {X 28.0774,Y 133.4878,Z 184,A 78.5372,B 3.7138,C 0.0591,E1 3.7515,E2 374.7429} C_DIS
LIN {X 32.082,Y 132.5804,Z 184,A 76.9463,B 3.7138,C 0.0592,E1 3.7558,E2 376.3172} C_DIS
LIN {X 35.6779,Y 131.6593,Z 184,A 75.336,B 3.7138,C 0.0609,E1 3.7602,E2 377.9333} C_DIS
LIN {X 40.6638,Y 130.2069,Z 184,A 73.2768,B 3.7137,C 0.0618,E1 3.7656,E2 379.9774} C_DIS
LIN {X 44.6429,Y 128.8944,Z 184,A 71.4183,B 3.7137,C 0.0644,E1 3.7706,E2 381.8472} C_DIS
LIN {X 48.6836,Y 127.4256,Z 184,A 69.7601,B 3.7137,C 0.065,E1 3.7749,E2 383.4875} C_DIS
LIN {X 51.3485,Y 126.3734,Z 184,A 68.5507,B 3.7137,C 0.0664,E1 3.778,E2 384.6973} C_DIS
LIN {X 54.3205,Y 125.1242,Z 184,A 67.2045,B 3.7136,C 0.0679,E1 3.7815,E2 386.0423} C_DIS
LIN {X 57.444,Y 123.7213,Z 184,A 65.7988,B 3.7136,C 0.0694,E1 3.785,E2 387.444} C_DIS
LIN {X 60.7964,Y 122.1097,Z 184,A 64.256,B 3.7136,C 0.0713,E1 3.7889,E2 388.9843} C_DIS
LIN {X 64.5833,Y 120.1511,Z 184,A 62.3286,B 3.7135,C 0.0751,E1 3.7937,E2 390.9281} C_DIS
LIN {X 67.7791,Y 118.3779,Z 184,A 60.8934,B 3.7135,C 0.0764,E1 3.7972,E2 392.3512} C_DIS
LIN {X 71.3591,Y 116.2547,Z 184,A 59.2056,B 3.7134,C 0.0784,E1 3.8012,E2 394.0317} C_DIS
LIN {X 75.0232,Y 113.9245,Z 184,A 57.4172,B 3.7134,C 0.081,E1 3.8054,E2 395.8157} C_DIS
LIN {X 78.7991,Y 111.3465,Z 184,A 55.551,B 3.7133,C 0.0837,E1 3.8096,E2 397.6755} C_DIS
LIN {X 82.3907,Y 108.7158,Z 184,A 53.7012,B 3.7132,C 0.0867,E1 3.8138,E2 399.5229} C_DIS
LIN {X 85.9314,Y 105.9397,Z 184,A 51.8462,B 3.7132,C 0.0898,E1 3.8178,E2 401.3738} C_DIS
LIN {X 89.3896,Y 103.0385,Z 184,A 49.9846,B 3.713,C 0.0931,E1 3.8218,E2 403.2314} C_DIS
LIN {X 95.1112,Y 97.7816,Z 184,A 47.0364,B 3.713,C 0.0963,E1 3.8277,E2 406.1416} C_DIS
LIN {X 97.2639,Y 95.6402,Z 184,A 45.2072,B 3.7127,C 0.1046,E1 3.8315,E2 408.0384} C_DIS
LIN {X 100.3003,Y 92.4509,Z 184,A 43.8253,B 3.7127,C 0.1037,E1 3.834,E2 409.3638} C_DIS
LIN {X 103.1983,Y 89.2045,Z 184,A 42.006,B 3.7127,C 0.1075,E1 3.8373,E2 411.1825} C_DIS
LIN {X 106.1952,Y 85.6146,Z 184,A 40.1494,B 3.7126,C 0.1108,E1 3.8406,E2 413.0264} C_DIS
LIN {X 108.8748,Y 82.18,Z 184,A 38.3488,B 3.7124,C 0.1146,E1 3.8437,E2 414.8239} C_DIS
LIN {X 111.6237,Y 78.4059,Z 184,A 36.4503,B 3.7124,C 0.1185,E1 3.8467,E2 416.7152} C_DIS
LIN {X 114.1119,Y 74.7387,Z 184,A 34.737,B 3.7122,C 0.1213,E1 3.8494,E2 418.4109} C_DIS
LIN {X 116.1807,Y 71.4798,Z 184,A 32.8807,B 3.712,C 0.1278,E1 3.8521,E2 420.2967} C_DIS
LIN {X 117.8766,Y 68.647,Z 184,A 31.7049,B 3.712,C 0.1289,E1 3.8538,E2 421.447} C_DIS
LIN {X 120.0931,Y 64.6912,Z 184,A 29.8963,B 3.7118,C 0.1326,E1 3.8562,E2 423.2445} C_DIS
LIN {X 122.2104,Y 60.5923,Z 184,A 28.1001,B 3.7118,C 0.136,E1 3.8584,E2 425.0239} C_DIS
LIN {X 123.8471,Y 57.172,Z 184,A 26.5355,B 3.7116,C 0.1398,E1 3.8603,E2 426.5857} C_DIS
LIN {X 125.487,Y 53.4814,Z 184,A 24.8134,B 3.7114,C 0.1445,E1 3.8622,E2 428.3118} C_DIS
LIN {X 127.739,Y 47.8486,Z 184,A 22.1537,B 3.7111,C 0.1524,E1 3.8649,E2 430.9864} C_DIS
LIN {X 128.9274,Y 44.5478,Z 184,A 21.0605,B 3.7111,C 0.1522,E1 3.8659,E2 432.0332} C_DIS
LIN {X 130.0065,Y 41.2932,Z 184,A 19.6677,B 3.711,C 0.1555,E1 3.8671,E2 433.4208} C_DIS
LIN {X 130.9948,Y 38.0425,Z 184,A 18.3089,B 3.7108,C 0.1587,E1 3.8682,E2 434.7718} C_DIS
LIN {X 131.904,Y 34.7605,Z 184,A 16.8575,B 3.7106,C 0.1628,E1 3.8692,E2 436.2267} C_DIS
LIN {X 132.9134,Y 30.6747,Z 184,A 15.1544,B 3.7105,C 0.1669,E1 3.8703,E2 437.9227} C_DIS
LIN {X 133.7407,Y 26.8396,Z 184,A 13.6067,B 3.7103,C 0.1704,E1 3.8712,E2 439.4588} C_DIS
LIN {X 134.4948,Y 22.7614,Z 184,A 11.8821,B 3.7101,C 0.175,E1 3.872,E2 441.1822} C_DIS
LIN {X 135.1405,Y 18.559,Z 184,A 9.9759,B 3.7098,C 0.1814,E1 3.8728,E2 443.1046} C_DIS
LIN {X 135.7687,Y 13.1814,Z 184,A 8.2824,B 3.7098,C 0.1813,E1 3.8733,E2 444.7265} C_DIS
LIN {X 136.31,Y 5.1468,Z 184,A 3.812,B 3.7087,C 0.203,E1 3.874,E2 449.3352} C_DIS
LIN {X 136.3937,Y -1.9394,Z 184,A 2.0941,B 3.709,C 0.1973,E1 3.874,E2 450.8977} C_DIS
LIN {X 136.194,Y -7.6544,Z 184,A -0.4687,B 3.7085,C 0.2059,E1 3.8737,E2 453.4827} C_DIS
LIN {X 135.7884,Y -12.9753,Z 184,A -2.9402,B 3.708,C 0.2148,E1 3.8731,E2 455.9846} C_DIS
LIN {X 135.3583,Y -16.8975,Z 184,A -4.2799,B 3.708,C 0.2159,E1 3.8727,E2 457.2855} C_DIS
LIN {X 134.7944,Y -20.9119,Z 184,A -5.7965,B 3.7078,C 0.2186,E1 3.8721,E2 458.7797} C_DIS
LIN {X 134.2188,Y -24.3359,Z 184,A -7.1918,B 3.7076,C 0.2219,E1 3.8714,E2 460.1682} C_DIS
LIN {X 133.5711,Y -27.6734,Z 184,A -8.5414,B 3.7074,C 0.225,E1 3.8707,E2 461.5088} C_DIS
LIN {X 132.9541,Y -30.4964,Z 184,A -9.7952,B 3.7072,C 0.2288,E1 3.8699,E2 462.7687} C_DIS
LIN {X 132.14,Y -33.8512,Z 184,A -11.1782,B 3.707,C 0.2321,E1 3.869,E2 464.1442} C_DIS
LIN {X 130.979,Y -38.0964,Z 184,A -12.9765,B 3.7067,C 0.2366,E1 3.8676,E2 465.9376} C_DIS
LIN {X 129.7448,Y -42.1125,Z 184,A -14.9978,B 3.7062,C 0.2442,E1 3.8659,E2 467.993} C_DIS
LIN {X 128.5373,Y -45.6654,Z 184,A -16.0743,B 3.7062,C 0.2429,E1 3.8649,E2 469.0071} C_DIS
LIN {X 126.9816,Y -49.8259,Z 184,A -18.0244,B 3.7059,C 0.2488,E1 3.863,E2 470.9694} C_DIS
LIN {X 125.0472,Y -54.4985,Z 184,A -19.9687,B 3.7056,C 0.2524,E1 3.8609,E2 472.8924} C_DIS
LIN {X 123.747,Y -57.3886,Z 184,A -21.3038,B 3.7054,C 0.2559,E1 3.8593,E2 474.2291} C_DIS
LIN {X 122.2082,Y -60.5966,Z 184,A -22.7344,B 3.7052,C 0.259,E1 3.8576,E2 475.6527} C_DIS
LIN {X 120.4522,Y -64.0191,Z 184,A -25.4755,B 3.704,C 0.2755,E1 3.8538,E2 478.5384} C_DIS
LIN {X 116.3307,Y -71.2353,Z 184,A -27.4022,B 3.7046,C 0.267,E1 3.8514,E2 480.2684} C_DIS
LIN {X 111.4163,Y -78.7,Z 184,A -31.3363,B 3.7038,C 0.2781,E1 3.8453,E2 484.2292} C_DIS
LIN {X 109.0229,Y -81.9838,Z 184,A -33.0646,B 3.7035,C 0.2822,E1 3.8423,E2 485.9618} C_DIS
LIN {X 106.2656,Y -85.5273,Z 184,A -34.8865,B 3.7032,C 0.2859,E1 3.8392,E2 487.777} C_DIS
LIN {X 103.6721,Y -88.654,Z 184,A -36.6276,B 3.7029,C 0.29,E1 3.836,E2 489.524} C_DIS
LIN {X 100.4979,Y -92.2359,Z 184,A -38.4423,B 3.7027,C 0.2923,E1 3.8327,E2 491.315} C_DIS
LIN {X 97.6263,Y -95.2707,Z 184,A -40.5817,B 3.7021,C 0.3001,E1 3.8284,E2 493.5056} C_DIS
LIN {X 94.5174,Y -98.3559,Z 184,A -41.8624,B 3.7023,C 0.2979,E1 3.826,E2 494.7156} C_DIS
LIN {X 90.6294,Y -101.9496,Z 184,A -44.1734,B 3.7018,C 0.3033,E1 3.8212,E2 497.0396} C_DIS
LIN {X 87.2091,Y -104.8901,Z 184,A -46.4392,B 3.7012,C 0.3108,E1 3.8163,E2 499.3549} C_DIS
LIN {X 83.5707,Y -107.811,Z 184,A -48.523,B 3.7008,C 0.3156,E1 3.8116,E2 501.4563} C_DIS
LIN {X 79.031,Y -111.1824,Z 184,A -50.0496,B 3.7012,C 0.3111,E1 3.8084,E2 502.875} C_DIS
LIN {X 76.2357,Y -113.1171,Z 184,A -51.61,B 3.7009,C 0.3148,E1 3.8048,E2 504.4537} C_DIS
LIN {X 72.4683,Y -115.5673,Z 184,A -53.3045,B 3.7008,C 0.316,E1 3.8008,E2 506.1245} C_DIS
LIN {X 68.9781,Y -117.6831,Z 184,A -55.3627,B 3.7002,C 0.3221,E1 3.7958,E2 508.2287} C_DIS
LIN {X 66.0138,Y -119.3712,Z 184,A -56.3239,B 3.7005,C 0.3195,E1 3.7936,E2 509.1297} C_DIS
LIN {X 63.3038,Y -120.8279,Z 184,A -57.7423,B 3.7002,C 0.3226,E1 3.79,E2 510.5655} C_DIS
LIN {X 59.9737,Y -122.5155,Z 184,A -59.3266,B 3.7,C 0.325,E1 3.7861,E2 512.153} C_DIS
LIN {X 56.8283,Y -124.006,Z 184,A -60.7013,B 3.6999,C 0.326,E1 3.7826,E2 513.5173} C_DIS
LIN {X 53.8753,Y -125.3167,Z 184,A -62.0256,B 3.6998,C 0.3274,E1 3.7792,E2 514.8384} C_DIS
LIN {X 50.8041,Y -126.5928,Z 184,A -63.4078,B 3.6996,C 0.3289,E1 3.7757,E2 516.2196} C_DIS
LIN {X 47.6544,Y -127.8118,Z 184,A -64.8066,B 3.6996,C 0.3303,E1 3.772,E2 517.6168} C_DIS
LIN {X 44.3861,Y -128.9835,Z 184,A -66.1569,B 3.6995,C 0.3309,E1 3.7685,E2 518.954} C_DIS
LIN {X 41.5114,Y -129.9368,Z 184,A -67.5426,B 3.6992,C 0.3332,E1 3.7648,E2 520.3553} C_DIS
LIN {X 37.5834,Y -131.1292,Z 184,A -69.1862,B 3.6992,C 0.3341,E1 3.7604,E2 521.9895} C_DIS
LIN {X 34.7518,Y -131.9063,Z 184,A -70.4625,B 3.699,C 0.3356,E1 3.7569,E2 523.2722} C_DIS
LIN {X 30.6285,Y -132.9239,Z 184,A -72.2185,B 3.699,C 0.3367,E1 3.7522,E2 525.0256} C_DIS
LIN {X 26.8501,Y -133.7386,Z 184,A -73.8015,B 3.6989,C 0.3375,E1 3.7478,E2 526.6043} C_DIS
LIN {X 21.8169,Y -134.6518,Z 184,A -76.1947,B 3.6985,C 0.3411,E1 3.7412,E2 529.0307} C_DIS
LIN {X 18.571,Y -135.1388,Z 184,A -77.258,B 3.6987,C 0.339,E1 3.7383,E2 530.0537} C_DIS
LIN {X 15.4084,Y -135.536,Z 184,A -79.4593,B 3.698,C 0.3473,E1 3.7319,E2 532.3678} C_DIS
LIN {X 9.1951,Y -136.0983,Z 184,A -81.1414,B 3.6986,C 0.34,E1 3.7276,E2 533.9293} C_DIS
LIN {X 5.0305,Y -136.3146,Z 184,A -83.2304,B 3.6983,C 0.3434,E1 3.7216,E2 536.0633} C_DIS
LIN {X 0.9677,Y -136.4022,Z 184,A -84.2911,B 3.6988,C 0.3382,E1 3.7189,E2 537.0403} C_DIS
Enddeposition()
LIN {X 0.9677,Y -136.4022,Z 184,A -84.2911,B 3.6988,C 0.3382,E1 3.7189,E2 537.0403} C_DIS
Startdeposition()
$VEL.CP = VEL_PRINT
LIN {X 2.2173,Y -137.29,Z 184,A -83.0628,B 3.6809,C 0.3334,E1 3.7042,E2 535.7539} C_DIS
LIN {X 6.2926,Y -137.1649,Z 184,A -81.5873,B 3.6807,C 0.3349,E1 3.7082,E2 534.3078} C_DIS
LIN {X 14.406,Y -136.5503,Z 184,A -78.3978,B 3.6807,C 0.3355,E1 3.717,E2 531.144} C_DIS
LIN {X 24.2644,Y -135.1467,Z 184,A -74.2266,B 3.6809,C 0.333,E1 3.7286,E2 526.9686} C_DIS
LIN {X 28.3268,Y -134.3556,Z 184,A -72.4681,B 3.6811,C 0.3315,E1 3.7334,E2 525.205} C_DIS
LIN {X 32.007,Y -133.5251,Z 184,A -70.9951,B 3.6811,C 0.3312,E1 3.7373,E2 523.7444} C_DIS
LIN {X 36.0061,Y -132.5041,Z 184,A -69.1697,B 3.6813,C 0.3287,E1 3.7423,E2 521.9043} C_DIS
LIN {X 39.9227,Y -131.3758,Z 184,A -67.6317,B 3.6813,C 0.3287,E1 3.7464,E2 520.3868} C_DIS
LIN {X 44.0987,Y -130.0355,Z 184,A -65.742,B 3.6815,C 0.3262,E1 3.7514,E2 518.488} C_DIS
LIN {X 47.9696,Y -128.6557,Z 184,A -64.2243,B 3.6815,C 0.3262,E1 3.7553,E2 516.9953} C_DIS
LIN {X 50.8499,Y -127.5456,Z 184,A -62.8345,B 3.6817,C 0.3238,E1 3.759,E2 515.5912} C_DIS
LIN {X 54.2055,Y -126.1554,Z 184,A -61.379,B 3.6819,C 0.3225,E1 3.7627,E2 514.1425} C_DIS
LIN {X 57.6902,Y -124.6,Z 184,A -59.8797,B 3.6819,C 0.3214,E1 3.7665,E2 512.6544} C_DIS
LIN {X 60.2343,Y -123.3915,Z 184,A -58.7661,B 3.682,C 0.3204,E1 3.7693,E2 511.5482} C_DIS
LIN {X 62.6105,Y -122.2021,Z 184,A -57.4448,B 3.6824,C 0.3167,E1 3.7727,E2 510.1978} C_DIS
LIN {X 66.6637,Y -120.041,Z 184,A -55.094,B 3.683,C 0.3095,E1 3.7786,E2 507.7877} C_DIS
LIN {X 71.0193,Y -117.5162,Z 184,A -53.6055,B 3.6827,C 0.3125,E1 3.7819,E2 506.3793} C_DIS
LIN {X 74.4549,Y -115.371,Z 184,A -51.8965,B 3.683,C 0.3095,E1 3.786,E2 504.6666} C_DIS
LIN {X 78.1247,Y -112.9182,Z 184,A -50.1914,B 3.6831,C 0.3079,E1 3.7899,E2 502.9782} C_DIS
LIN {X 81.6851,Y -110.3701,Z 184,A -48.2776,B 3.6834,C 0.3037,E1 3.7942,E2 501.0515} C_DIS
LIN {X 85.3591,Y -107.5534,Z 184,A -46.3254,B 3.6838,C 0.3,E1 3.7985,E2 499.095} C_DIS
LIN {X 89.2816,Y -104.3208,Z 184,A -44.3541,B 3.684,C 0.2975,E1 3.8027,E2 497.1418} C_DIS
LIN {X 92.6522,Y -101.3389,Z 184,A -42.5327,B 3.6842,C 0.2944,E1 3.8065,E2 495.3264} C_DIS
LIN {X 95.7616,Y -98.4057,Z 184,A -40.7218,B 3.6845,C 0.2905,E1 3.8101,E2 493.5105} C_DIS
LIN {X 99.1323,Y -95.0088,Z 184,A -38.8352,B 3.6848,C 0.2875,E1 3.8138,E2 491.6369} C_DIS
LIN {X 104.015,Y -89.6367,Z 184,A -36.1332,B 3.685,C 0.2845,E1 3.8188,E2 488.9756} C_DIS
LIN {X 106.4931,Y -86.6785,Z 184,A -34.321,B 3.6854,C 0.2786,E1 3.822,E2 487.1354} C_DIS
LIN {X 109.3242,Y -83.0798,Z 184,A -32.4969,B 3.6857,C 0.2752,E1 3.8251,E2 485.3212} C_DIS
LIN {X 111.9511,Y -79.5047,Z 184,A -30.8895,B 3.6858,C 0.2735,E1 3.8277,E2 483.7444} C_DIS
LIN {X 114.8266,Y -75.2912,Z 184,A -28.6895,B 3.6862,C 0.2677,E1 3.8312,E2 481.5332} C_DIS
LIN {X 117.1634,Y -71.6007,Z 184,A -26.8686,B 3.6866,C 0.2632,E1 3.8339,E2 479.711} C_DIS
LIN {X 118.8265,Y -68.805,Z 184,A -25.2509,B 3.687,C 0.2569,E1 3.8362,E2 478.058} C_DIS
LIN {X 120.7892,Y -65.2988,Z 184,A -23.8986,B 3.687,C 0.2563,E1 3.8379,E2 476.7471} C_DIS
LIN {X 122.958,Y -61.1131,Z 184,A -22.1113,B 3.6873,C 0.2533,E1 3.8402,E2 474.9817} C_DIS
LIN {X 124.5071,Y -57.891,Z 184,A -20.7108,B 3.6874,C 0.2505,E1 3.8418,E2 473.5918} C_DIS
LIN {X 126.3465,Y -53.7634,Z 184,A -18.7113,B 3.6879,C 0.2443,E1 3.8441,E2 471.576} C_DIS
LIN {X 127.839,Y -50.1064,Z 184,A -17.4506,B 3.6879,C 0.2443,E1 3.8453,E2 470.3645} C_DIS
LIN {X 129.1246,Y -46.6926,Z 184,A -15.9178,B 3.6881,C 0.2401,E1 3.8468,E2 468.8291} C_DIS
LIN {X 129.9776,Y -44.2689,Z 184,A -14.7424,B 3.6884,C 0.236,E1 3.8479,E2 467.6395} C_DIS
LIN {X 131.0869,Y -40.8666,Z 184,A -13.2532,B 3.6887,C 0.232,E1 3.8492,E2 466.1496} C_DIS
LIN {X 132.1879,Y -37.1448,Z 184,A -11.8026,B 3.6888,C 0.2295,E1 3.8503,E2 464.7197} C_DIS
LIN {X 132.9542,Y -34.3053,Z 184,A -10.707,B 3.6889,C 0.2277,E1 3.851,E2 463.6403} C_DIS
LIN {X 133.7653,Y -30.9905,Z 184,A -9.3771,B 3.6891,C 0.2248,E1 3.8519,E2 462.3214} C_DIS
LIN {X 134.4844,Y -27.7027,Z 184,A -7.8503,B 3.6894,C 0.2195,E1 3.8528,E2 460.7777} C_DIS
LIN {X 135.1703,Y -24.1325,Z 184,A -6.411,B 3.6896,C 0.2162,E1 3.8535,E2 459.3473} C_DIS
LIN {X 135.7942,Y -20.3423,Z 184,A -4.3471,B 3.6902,C 0.2064,E1 3.8544,E2 457.2223} C_DIS
LIN {X 136.3989,Y -15.7799,Z 184,A -3.0461,B 3.6901,C 0.2081,E1 3.8548,E2 456.0004} C_DIS
LIN {X 136.7339,Y -12.5539,Z 184,A -1.5799,B 3.6904,C 0.203,E1 3.8552,E2 454.5186} C_DIS
LIN {X 137.0242,Y -8.8303,Z 184,A -0.2554,B 3.6904,C 0.2013,E1 3.8555,E2 453.2232} C_DIS
LIN {X 137.2846,Y -2.5464,Z 184,A 2.6295,B 3.691,C 0.1909,E1 3.8557,E2 450.303} C_DIS
LIN {X 137.3048,Y 0.9383,Z 184,A 3.6945,B 3.691,C 0.1912,E1 3.8557,E2 449.2871} C_DIS
LIN {X 137.2181,Y 4.98,Z 184,A 5.2552,B 3.6912,C 0.1879,E1 3.8557,E2 447.7415} C_DIS
LIN {X 136.775,Y 12.0963,Z 184,A 8.1814,B 3.6915,C 0.1801,E1 3.8551,E2 444.8199} C_DIS
LIN {X 135.9735,Y 19.0976,Z 184,A 11.0696,B 3.6919,C 0.1724,E1 3.8541,E2 441.9366} C_DIS
LIN {X 135.5503,Y 21.9093,Z 184,A 12.1204,B 3.6919,C 0.1706,E1 3.8536,E2 440.9025} C_DIS
LIN {X 134.9152,Y 25.5216,Z 184,A 13.637,B 3.6922,C 0.1665,E1 3.8529,E2 439.3868} C_DIS
LIN {X 134.3377,Y 28.4094,Z 184,A 14.737,B 3.6922,C 0.1646,E1 3.8523,E2 438.3025} C_DIS
LIN {X 133.5528,Y 31.8919,Z 184,A 16.3009,B 3.6925,C 0.1596,E1 3.8513,E2 436.7282} C_DIS
LIN {X 132.7134,Y 35.2213,Z 184,A 17.6478,B 3.6926,C 0.1567,E1 3.8503,E2 435.3915} C_DIS
LIN {X 131.8292,Y 38.3986,Z 184,A 18.8696,B 3.6926,C 0.1547,E1 3.8494,E2 434.1886} C_DIS
LIN {X 130.893,Y 41.4784,Z 184,A 20.288,B 3.6929,C 0.1502,E1 3.8482,E2 432.76} C_DIS
LIN {X 129.5908,Y 45.3845,Z 184,A 23.1418,B 3.6935,C 0.1329,E1 3.8455,E2 429.7599} C_DIS
LIN {X 126.5244,Y 53.3396,Z 184,A 25.1873,B 3.6933,C 0.1404,E1 3.8435,E2 427.9062} C_DIS
LIN {X 124.4818,Y 57.9458,Z 184,A 27.5103,B 3.6936,C 0.1325,E1 3.8408,E2 425.5545} C_DIS
LIN {X 122.6515,Y 61.7278,Z 184,A 29.1662,B 3.6936,C 0.1291,E1 3.8388,E2 423.9103} C_DIS
LIN {X 120.7247,Y 65.4183,Z 184,A 30.798,B 3.6938,C 0.1259,E1 3.8366,E2 422.2911} C_DIS
LIN {X 116.7145,Y 72.3301,Z 184,A 33.9528,B 3.694,C 0.1197,E1 3.8322,E2 419.1579} C_DIS
LIN {X 114.2895,Y 76.1038,Z 184,A 35.9093,B 3.6942,C 0.1143,E1 3.8292,E2 417.1902} C_DIS
LIN {X 111.7277,Y 79.8172,Z 184,A 37.7236,B 3.6942,C 0.1107,E1 3.8263,E2 415.3838} C_DIS
LIN {X 108.946,Y 83.5743,Z 184,A 39.5331,B 3.6944,C 0.1077,E1 3.8233,E2 413.5915} C_DIS
LIN {X 106.5152,Y 86.6513,Z 184,A 41.2337,B 3.6944,C 0.1034,E1 3.8203,E2 411.8825} C_DIS
LIN {X 103.5047,Y 90.2255,Z 184,A 43.0749,B 3.6946,C 0.1003,E1 3.817,E2 410.0544} C_DIS
LIN {X 100.0846,Y 94.0054,Z 184,A 45.1824,B 3.6946,C 0.096,E1 3.813,E2 407.949} C_DIS
LIN {X 96.9401,Y 97.2446,Z 184,A 46.7874,B 3.6947,C 0.095,E1 3.8099,E2 406.3784} C_DIS
LIN {X 94.6065,Y 99.5168,Z 184,A 48.1216,B 3.6947,C 0.0925,E1 3.8072,E2 405.0471} C_DIS
LIN {X 91.9232,Y 102.0008,Z 184,A 49.8499,B 3.6949,C 0.0875,E1 3.8036,E2 403.2934} C_DIS
LIN {X 88.4171,Y 105.0538,Z 184,A 51.6764,B 3.6949,C 0.0849,E1 3.7998,E2 401.4809} C_DIS
LIN {X 85.0888,Y 107.7677,Z 184,A 53.4755,B 3.695,C 0.0816,E1 3.7958,E2 399.6807} C_DIS
LIN {X 81.4956,Y 110.5097,Z 184,A 55.3058,B 3.695,C 0.0789,E1 3.7918,E2 397.8573} C_DIS
LIN {X 77.8117,Y 113.1336,Z 184,A 57.1355,B 3.6951,C 0.0763,E1 3.7876,E2 396.0347} C_DIS
LIN {X 73.9371,Y 115.703,Z 184,A 58.9943,B 3.6951,C 0.074,E1 3.7833,E2 394.1859} C_DIS
LIN {X 70.6277,Y 117.7528,Z 184,A 60.5904,B 3.6952,C 0.0718,E1 3.7795,E2 392.5934} C_DIS
LIN {X 67.1656,Y 119.7609,Z 184,A 62.1782,B 3.6952,C 0.0701,E1 3.7756,E2 391.0159} C_DIS
LIN {X 64.0144,Y 121.4722,Z 184,A 63.6318,B 3.6952,C 0.0684,E1 3.7721,E2 389.5675} C_DIS
LIN {X 61.0675,Y 122.9804,Z 184,A 64.866,B 3.6953,C 0.0679,E1 3.769,E2 388.3516} C_DIS
LIN {X 58.5609,Y 124.1951,Z 184,A 66.128,B 3.6953,C 0.0655,E1 3.7658,E2 387.0774} C_DIS
LIN {X 54.918,Y 125.8473,Z 184,A 67.7973,B 3.6953,C 0.0635,E1 3.7616,E2 385.4083} C_DIS
LIN {X 51.5317,Y 127.2708,Z 184,A 69.197,B 3.6953,C 0.0629,E1 3.758,E2 384.0252} C_DIS
LIN {X 48.9245,Y 128.298,Z 184,A 70.4156,B 3.6954,C 0.0612,E1 3.7548,E2 382.8009} C_DIS
LIN {X 45.4309,Y 129.5747,Z 184,A 71.9348,B 3.6954,C 0.0599,E1 3.7508,E2 381.2859} C_DIS
LIN {X 42.6191,Y 130.5281,Z 184,A 73.173,B 3.6954,C 0.0587,E1 3.7475,E2 380.0481} C_DIS
LIN {X 40.1526,Y 131.3054,Z 184,A 74.3258,B 3.6954,C 0.057,E1 3.7444,E2 378.8864} C_DIS
LIN {X 35.7818,Y 132.5639,Z 184,A 76.1732,B 3.6955,C 0.0559,E1 3.7395,E2 377.0457} C_DIS
LIN {X 32.2819,Y 133.4589,Z 184,A 77.6075,B 3.6955,C 0.0554,E1 3.7356,E2 375.6207} C_DIS
LIN {X 29.1608,Y 134.1755,Z 184,A 78.8372,B 3.6955,C 0.0554,E1 3.7323,E2 374.4044} C_DIS
LIN {X 26.5839,Y 134.7121,Z 184,A 80.1802,B 3.6955,C 0.0525,E1 3.7285,E2 373.0319} C_DIS
LIN {X 22.6618,Y 135.4247,Z 184,A 81.6852,B 3.6955,C 0.0529,E1 3.7244,E2 371.5467} C_DIS
LIN {X 18.6536,Y 136.0368,Z 184,A 83.7591,B 3.6956,C 0.0489,E1 3.7186,E2 369.4265} C_DIS
LIN {X 14.9329,Y 136.4936,Z 184,A 85.3847,B 3.6956,C 0.0477,E1 3.714,E2 367.7938} C_DIS
LIN {X 10.6176,Y 136.8981,Z 184,A 86.707,B 3.6956,C 0.0512,E1 3.7105,E2 366.5321} C_DIS
LIN {X 3.3111,Y 137.2689,Z 184,A 89.7183,B 3.6956,C 0.0509,E1 3.7021,E2 363.5272} C_DIS
LIN {X -4.8234,Y 137.2242,Z 184,A 94.3391,B 3.6957,C 0.0409,E1 3.6888,E2 358.7563} C_DIS
LIN {X -12.8798,Y 136.7026,Z 184,A 96.728,B 3.6957,C 0.0491,E1 3.6825,E2 356.4906} C_DIS
LIN {X -17.2769,Y 136.2177,Z 184,A 98.4536,B 3.6956,C 0.0505,E1 3.6777,E2 354.7808} C_DIS
LIN {X -21.0519,Y 135.6843,Z 184,A 100.011,B 3.6956,C 0.0513,E1 3.6735,E2 353.2283} C_DIS
LIN {X -24.6996,Y 135.0688,Z 184,A 101.6334,B 3.6956,C 0.0513,E1 3.669,E2 351.597} C_DIS
LIN {X -28.5481,Y 134.3078,Z 184,A 103.0484,B 3.6956,C 0.0537,E1 3.6652,E2 350.2101} C_DIS
LIN {X -31.841,Y 133.5651,Z 184,A 104.5986,B 3.6956,C 0.0535,E1 3.6609,E2 348.6434} C_DIS
LIN {X -35.2508,Y 132.7056,Z 184,A 106.0806,B 3.6956,C 0.0543,E1 3.6569,E2 347.1605} C_DIS
LIN {X -38.3001,Y 131.858,Z 184,A 107.2912,B 3.6956,C 0.056,E1 3.6537,E2 345.964} C_DIS
LIN {X -40.7556,Y 131.1209,Z 184,A 108.5869,B 3.6956,C 0.0552,E1 3.6501,E2 344.6415} C_DIS
LIN {X -44.7149,Y 129.8229,Z 184,A 110.3254,B 3.6955,C 0.0566,E1 3.6455,E2 342.904} C_DIS
LIN {X -47.8737,Y 128.6916,Z 184,A 111.5248,B 3.6955,C 0.0592,E1 3.6425,E2 341.73} C_DIS
LIN {X -50.2651,Y 127.7774,Z 184,A 112.9968,B 3.6955,C 0.0575,E1 3.6385,E2 340.2093} C_DIS
LIN {X -54.2498,Y 126.1362,Z 184,A 114.5405,B 3.6955,C 0.061,E1 3.6346,E2 338.6979} C_DIS
LIN {X -57.43,Y 124.7203,Z 184,A 116.0286,B 3.6955,C 0.0624,E1 3.6308,E2 337.2065} C_DIS
LIN {X -60.6029,Y 123.2096,Z 184,A 118.1728,B 3.6955,C 0.0596,E1 3.6252,E2 334.9797} C_DIS
LIN {X -65.2126,Y 120.8356,Z 184,A 119.8401,B 3.6954,C 0.0656,E1 3.6213,E2 333.3753} C_DIS
LIN {X -68.7228,Y 118.874,Z 184,A 121.7872,B 3.6954,C 0.0661,E1 3.6165,E2 331.3962} C_DIS
LIN {X -71.7274,Y 117.0856,Z 184,A 122.9682,B 3.6953,C 0.0699,E1 3.6137,E2 330.2506} C_DIS
LIN {X -75.0896,Y 114.959,Z 184,A 124.7576,B 3.6953,C 0.0715,E1 3.6095,E2 328.4465} C_DIS
LIN {X -78.9137,Y 112.368,Z 184,A 126.68,B 3.6952,C 0.0745,E1 3.6051,E2 326.5261} C_DIS
LIN {X -82.2248,Y 109.9682,Z 184,A 128.2868,B 3.6952,C 0.0779,E1 3.6015,E2 324.9328} C_DIS
LIN {X -85.6508,Y 107.3212,Z 184,A 130.285,B 3.6951,C 0.0798,E1 3.597,E2 322.9124} C_DIS
LIN {X -89.1472,Y 104.4352,Z 184,A 132.2529,B 3.6951,C 0.0827,E1 3.5928,E2 320.9365} C_DIS
LIN {X -92.3572,Y 101.6072,Z 184,A 134.0413,B 3.6949,C 0.0859,E1 3.5891,E2 319.149} C_DIS
LIN {X -95.4889,Y 98.6698,Z 184,A 135.9789,B 3.6949,C 0.0885,E1 3.5852,E2 317.1948} C_DIS
LIN {X -98.8943,Y 95.257,Z 184,A 138.0158,B 3.6948,C 0.0923,E1 3.5812,E2 315.1565} C_DIS
LIN {X -101.7401,Y 92.2107,Z 184,A 139.7785,B 3.6947,C 0.0957,E1 3.5778,E2 313.3922} C_DIS
LIN {X -104.6515,Y 88.8927,Z 184,A 141.7972,B 3.6947,C 0.0986,E1 3.5741,E2 311.3531} C_DIS
LIN {X -107.9571,Y 84.8477,Z 184,A 143.9115,B 3.6945,C 0.1037,E1 3.5704,E2 309.2486} C_DIS
LIN {X -110.7449,Y 81.1754,Z 184,A 145.8641,B 3.6944,C 0.1079,E1 3.5672,E2 307.2939} C_DIS
LIN {X -113.2908,Y 77.5827,Z 184,A 147.7626,B 3.6942,C 0.1117,E1 3.5641,E2 305.3893} C_DIS
LIN {X -115.9927,Y 73.482,Z 184,A 149.9179,B 3.6942,C 0.116,E1 3.5609,E2 303.2225} C_DIS
LIN {X -118.3507,Y 69.6202,Z 184,A 151.8321,B 3.694,C 0.1204,E1 3.5581,E2 301.3065} C_DIS
LIN {X -120.4591,Y 65.9053,Z 184,A 153.6901,B 3.6938,C 0.1244,E1 3.5556,E2 299.4406} C_DIS
LIN {X -122.1202,Y 62.7714,Z 184,A 155.1976,B 3.6938,C 0.1279,E1 3.5536,E2 297.9308} C_DIS
LIN {X -123.761,Y 59.4695,Z 184,A 156.5694,B 3.6936,C 0.1327,E1 3.552,E2 296.581} C_DIS
LIN {X -127.2496,Y 51.5841,Z 184,A 160.5562,B 3.6933,C 0.14,E1 3.5475,E2 292.5488} C_DIS
LIN {X -128.4971,Y 48.3929,Z 184,A 161.7944,B 3.6931,C 0.1447,E1 3.5462,E2 291.3356} C_DIS
LIN {X -129.566,Y 45.4561,Z 184,A 163.4119,B 3.6931,C 0.1466,E1 3.5447,E2 289.68} C_DIS
LIN {X -130.8509,Y 41.6102,Z 184,A 164.9741,B 3.6928,C 0.1518,E1 3.5434,E2 288.1353} C_DIS
LIN {X -131.8298,Y 38.3964,Z 184,A 166.6054,B 3.6928,C 0.1544,E1 3.542,E2 286.4763} C_DIS
LIN {X -132.9708,Y 34.2399,Z 184,A 168.5083,B 3.6925,C 0.1588,E1 3.5407,E2 284.5617} C_DIS
LIN {X -134.0852,Y 29.579,Z 184,A 170.6295,B 3.6923,C 0.1637,E1 3.5393,E2 282.4267} C_DIS
LIN {X -135.0142,Y 25.0036,Z 184,A 172.6308,B 3.6921,C 0.1688,E1 3.5383,E2 280.4201} C_DIS
LIN {X -135.6834,Y 21.0579,Z 184,A 174.3082,B 3.6919,C 0.1734,E1 3.5375,E2 278.743} C_DIS
LIN {X -136.234,Y 17.1526,Z 184,A 176.069,B 3.6917,C 0.1775,E1 3.5369,E2 276.9689} C_DIS
LIN {X -136.6991,Y 12.9167,Z 184,A 177.8273,B 3.6914,C 0.1825,E1 3.5364,E2 275.2144} C_DIS
LIN {X -137.033,Y 8.6871,Z 184,A 179.6694,B 3.6912,C 0.1872,E1 3.536,E2 273.3644} C_DIS
LIN {X -137.2311,Y 4.6464,Z 184,A -178.6398,B 3.691,C 0.1919,E1 3.5358,E2 271.6745} C_DIS
LIN {X -137.3048,Y 0.9348,Z 184,A -176.9089,B 3.6908,C 0.1954,E1 3.5358,E2 269.9215} C_DIS
LIN {X -137.2618,Y -3.5687,Z 184,A -175.0186,B 3.6905,C 0.2006,E1 3.5358,E2 268.031} C_DIS
LIN {X -137.1331,Y -6.9252,Z 184,A -173.5282,B 3.6903,C 0.2041,E1 3.536,E2 266.5302} C_DIS
LIN {X -136.8497,Y -11.2119,Z 184,A -171.8758,B 3.69,C 0.2099,E1 3.5364,E2 264.8969} C_DIS
LIN {X -136.5298,Y -14.5965,Z 184,A -170.2087,B 3.6898,C 0.2126,E1 3.5368,E2 263.1989} C_DIS
LIN {X -136.0439,Y -18.6026,Z 184,A -168.3524,B 3.6896,C 0.2164,E1 3.5375,E2 261.3217} C_DIS
LIN {X -135.4611,Y -22.4434,Z 184,A -166.8512,B 3.6893,C 0.2216,E1 3.5381,E2 259.8367} C_DIS
LIN {X -134.9855,Y -25.1536,Z 184,A -165.5039,B 3.6892,C 0.2237,E1 3.5388,E2 258.4647} C_DIS
LIN {X -134.2538,Y -28.7982,Z 184,A -164.0129,B 3.6889,C 0.2283,E1 3.5397,E2 256.9822} C_DIS
LIN {X -133.2722,Y -33.0521,Z 184,A -162.0416,B 3.6886,C 0.2325,E1 3.541,E2 254.9928} C_DIS
LIN {X -132.5081,Y -35.9911,Z 184,A -160.6494,B 3.6884,C 0.2353,E1 3.542,E2 253.5852} C_DIS
LIN {X -131.358,Y -39.9808,Z 184,A -159.0046,B 3.6881,C 0.2404,E1 3.5433,E2 251.9525} C_DIS
LIN {X -130.517,Y -42.6527,Z 184,A -157.5896,B 3.688,C 0.2422,E1 3.5445,E2 250.5065} C_DIS
LIN {X -129.3233,Y -46.1413,Z 184,A -156.2971,B 3.6876,C 0.2476,E1 3.5457,E2 249.2464} C_DIS
LIN {X -128.2512,Y -49.0461,Z 184,A -154.7018,B 3.6876,C 0.2493,E1 3.5473,E2 247.6126} C_DIS
LIN {X -126.8327,Y -52.6014,Z 184,A -153.1724,B 3.6872,C 0.2538,E1 3.5489,E2 246.0927} C_DIS
LIN {X -125.338,Y -56.0687,Z 184,A -151.6185,B 3.6869,C 0.258,E1 3.5506,E2 244.5423} C_DIS
LIN {X -123.9413,Y -59.092,Z 184,A -150.1272,B 3.6867,C 0.2609,E1 3.5524,E2 243.0384} C_DIS
LIN {X -122.4372,Y -62.1487,Z 184,A -148.6063,B 3.6865,C 0.2639,E1 3.5543,E2 241.5052} C_DIS
LIN {X -120.7364,Y -65.3969,Z 184,A -146.9075,B 3.6863,C 0.2667,E1 3.5566,E2 239.7852} C_DIS
LIN {X -118.9777,Y -68.5438,Z 184,A -145.3736,B 3.6861,C 0.2702,E1 3.5587,E2 238.248} C_DIS
LIN {X -116.6413,Y -72.4478,Z 184,A -143.4249,B 3.6857,C 0.2743,E1 3.5616,E2 236.2934} C_DIS
LIN {X -114.1203,Y -76.3574,Z 184,A -141.4339,B 3.6854,C 0.2785,E1 3.5646,E2 234.2965} C_DIS
LIN {X -111.5041,Y -80.1299,Z 184,A -139.4577,B 3.6851,C 0.2825,E1 3.5678,E2 232.313} C_DIS
LIN {X -108.9401,Y -83.582,Z 184,A -137.6252,B 3.6849,C 0.2862,E1 3.5709,E2 230.476} C_DIS
LIN {X -106.1256,Y -87.1281,Z 184,A -135.6378,B 3.6846,C 0.2896,E1 3.5744,E2 228.4762} C_DIS
LIN {X -103.2737,Y -90.4903,Z 184,A -132.9635,B 3.6846,C 0.2882,E1 3.5796,E2 225.6922} C_DIS
LIN {X -98.9377,Y -95.2122,Z 184,A -131.2762,B 3.6838,C 0.2997,E1 3.5826,E2 224.1357} C_DIS
LIN {X -96.0539,Y -98.12,Z 184,A -129.2725,B 3.6837,C 0.3011,E1 3.5866,E2 222.0936} C_DIS
LIN {X -92.7398,Y -101.2583,Z 184,A -127.2973,B 3.6834,C 0.3041,E1 3.5906,E2 220.1094} C_DIS
LIN {X -89.3496,Y -104.2623,Z 184,A -125.3478,B 3.6832,C 0.3071,E1 3.5948,E2 218.1522} C_DIS
LIN {X -85.877,Y -107.1409,Z 184,A -123.4046,B 3.6829,C 0.3099,E1 3.599,E2 216.2012} C_DIS
LIN {X -82.3631,Y -109.8652,Z 184,A -121.5365,B 3.6827,C 0.3128,E1 3.6032,E2 214.3315} C_DIS
LIN {X -78.8769,Y -112.3939,Z 184,A -119.6968,B 3.6825,C 0.3152,E1 3.6074,E2 212.4862} C_DIS
LIN {X -75.1471,Y -114.9215,Z 184,A -117.7914,B 3.6823,C 0.3178,E1 3.6118,E2 210.5775} C_DIS
LIN {X -71.7483,Y -117.0728,Z 184,A -116.1363,B 3.682,C 0.3202,E1 3.6157,E2 208.9254} C_DIS
LIN {X -67.9891,Y -119.2952,Z 184,A -114.2284,B 3.6819,C 0.322,E1 3.6203,E2 207.006} C_DIS
LIN {X -64.1772,Y -121.3867,Z 184,A -112.5754,B 3.6816,C 0.3254,E1 3.6244,E2 205.3741} C_DIS
LIN {X -61.6921,Y -122.6696,Z 184,A -111.2807,B 3.6816,C 0.3258,E1 3.6276,E2 204.0625} C_DIS
LIN {X -58.0457,Y -124.4356,Z 184,A -109.5309,B 3.6814,C 0.3272,E1 3.6321,E2 202.3046} C_DIS
LIN {X -54.8332,Y -125.884,Z 184,A -108.1004,B 3.6813,C 0.329,E1 3.6357,E2 200.8792} C_DIS
LIN {X -52.0594,Y -127.0581,Z 184,A -106.827,B 3.6812,C 0.3301,E1 3.639,E2 199.6034} C_DIS
LIN {X -48.8375,Y -128.3306,Z 184,A -105.2771,B 3.6812,C 0.3306,E1 3.6431,E2 198.0395} C_DIS
LIN {X -45.8187,Y -129.4396,Z 184,A -103.9881,B 3.681,C 0.3321,E1 3.6464,E2 196.7572} C_DIS
LIN {X -43.1592,Y -130.3483,Z 184,A -102.9054,B 3.6809,C 0.3336,E1 3.6493,E2 195.6861} C_DIS
LIN {X -40.4434,Y -131.2165,Z 184,A -101.6131,B 3.6809,C 0.3336,E1 3.6528,E2 194.3799} C_DIS
LIN {X -37.1343,Y -132.1909,Z 184,A -100.1339,B 3.6809,C 0.3343,E1 3.6568,E2 192.8951} C_DIS
LIN {X -34.0093,Y -133.0293,Z 184,A -98.7545,B 3.6808,C 0.3348,E1 3.6605,E2 191.5114} C_DIS
LIN {X -30.95,Y -133.7745,Z 184,A -97.5769,B 3.6806,C 0.3366,E1 3.6637,E2 190.3515} C_DIS
LIN {X -28.085,Y -134.4066,Z 184,A -96.1074,B 3.6807,C 0.3352,E1 3.6678,E2 188.8491} C_DIS
LIN {X -24.2351,Y -135.152,Z 184,A -94.7043,B 3.6805,C 0.3377,E1 3.6715,E2 187.4764} C_DIS
LIN {X -19.2728,Y -135.9485,Z 184,A -92.4497,B 3.6805,C 0.337,E1 3.6778,E2 185.2002} C_DIS
LIN {X -15.4682,Y -136.436,Z 184,A -90.7413,B 3.6806,C 0.3364,E1 3.6826,E2 183.4769} C_DIS
LIN {X -11.7774,Y -136.802,Z 184,A -89.0123,B 3.6807,C 0.335,E1 3.6875,E2 181.723} C_DIS
LIN {X -8.4225,Y -137.0493,Z 184,A -87.7948,B 3.6806,C 0.3366,E1 3.6908,E2 180.5296} C_DIS
LIN {X -3.761,Y -137.2564,Z 184,A -85.9438,B 3.6806,C 0.3373,E1 3.6959,E2 178.6906} C_DIS
LIN {X 0.4514,Y -137.3076,Z 184,A -84.1941,B 3.6806,C 0.3372,E1 3.7008,E2 176.9412} C_DIS
LIN {X 0.4514,Y -137.3076,Z 184,A -84.1941,B 3.6806,C 0.3372,E1 3.7008,E2 176.9412} C_DIS
Enddeposition()
LIN {X 0.9865,Y -138.204,Z 184,A -84.0712,B 3.6624,C 0.3395,E1 3.6832,E2 176.8676} C_DIS
Startdeposition()
$VEL.CP = VEL_PRINT
LIN {X -3.0237,Y -138.1776,Z 184,A -86.2078,B 3.662,C 0.3438,E1 3.677,E2 179.0684} C_DIS
LIN {X -6.1171,Y -138.0752,Z 184,A -87.4927,B 3.662,C 0.3438,E1 3.6734,E2 180.3541} C_DIS
LIN {X -9.2792,Y -137.8991,Z 184,A -88.8078,B 3.662,C 0.3438,E1 3.6698,E2 181.6701} C_DIS
LIN {X -13.3553,Y -137.5619,Z 184,A -90.5403,B 3.662,C 0.344,E1 3.6649,E2 183.4082} C_DIS
LIN {X -17.1189,Y -137.1464,Z 184,A -92.0861,B 3.662,C 0.3435,E1 3.6606,E2 184.9514} C_DIS
LIN {X -20.3485,Y -136.7048,Z 184,A -93.4436,B 3.662,C 0.3432,E1 3.6569,E2 186.3102} C_DIS
LIN {X -23.5462,Y -136.1904,Z 184,A -94.7944,B 3.662,C 0.3429,E1 3.6532,E2 187.6626} C_DIS
LIN {X -26.1972,Y -135.7032,Z 184,A -95.9703,B 3.662,C 0.3429,E1 3.6499,E2 188.8465} C_DIS
LIN {X -29.9253,Y -134.932,Z 184,A -97.5098,B 3.6622,C 0.3419,E1 3.6457,E2 190.3815} C_DIS
LIN {X -33.1472,Y -134.1769,Z 184,A -98.8936,B 3.6622,C 0.3413,E1 3.6419,E2 191.7673} C_DIS
LIN {X -35.9002,Y -133.4647,Z 184,A -100.0836,B 3.6622,C 0.3407,E1 3.6387,E2 192.959} C_DIS
LIN {X -39.3824,Y -132.4798,Z 184,A -101.6112,B 3.6624,C 0.3399,E1 3.6346,E2 194.4907} C_DIS
LIN {X -42.647,Y -131.4654,Z 184,A -103.0425,B 3.6624,C 0.339,E1 3.6308,E2 195.9242} C_DIS
LIN {X -46.0747,Y -130.3049,Z 184,A -104.5513,B 3.6626,C 0.3379,E1 3.6268,E2 197.4345} C_DIS
LIN {X -49.1625,Y -129.1709,Z 184,A -105.9348,B 3.6626,C 0.3369,E1 3.6232,E2 198.8209} C_DIS
LIN {X -52.4222,Y -127.8831,Z 184,A -107.4062,B 3.6628,C 0.3357,E1 3.6193,E2 200.295} C_DIS
LIN {X -55.5957,Y -126.5358,Z 184,A -108.8527,B 3.6628,C 0.3344,E1 3.6156,E2 201.744} C_DIS
LIN {X -58.3461,Y -125.2892,Z 184,A -110.1696,B 3.6629,C 0.3336,E1 3.6123,E2 203.0696} C_DIS
LIN {X -61.8796,Y -123.5843,Z 184,A -111.7819,B 3.6631,C 0.3317,E1 3.6082,E2 204.6803} C_DIS
LIN {X -64.9833,Y -121.9809,Z 184,A -113.0841,B 3.6634,C 0.3289,E1 3.605,E2 205.9633} C_DIS
LIN {X -67.6738,Y -120.5086,Z 184,A -114.6264,B 3.6634,C 0.3292,E1 3.6012,E2 207.5414} C_DIS
LIN {X -71.4307,Y -118.3205,Z 184,A -116.4712,B 3.6635,C 0.3272,E1 3.5967,E2 209.392} C_DIS
LIN {X -74.8883,Y -116.1637,Z 184,A -118.186,B 3.6637,C 0.325,E1 3.5927,E2 211.1102} C_DIS
LIN {X -78.551,Y -113.7188,Z 184,A -119.9762,B 3.664,C 0.322,E1 3.5886,E2 212.8958} C_DIS
LIN {X -81.4686,Y -111.6473,Z 184,A -121.4928,B 3.6642,C 0.32,E1 3.5851,E2 214.4166} C_DIS
LIN {X -84.2967,Y -109.5276,Z 184,A -123.1059,B 3.6642,C 0.3186,E1 3.5815,E2 216.0491} C_DIS
LIN {X -87.805,Y -106.7359,Z 184,A -124.8927,B 3.6646,C 0.315,E1 3.5776,E2 217.8263} C_DIS
LIN {X -90.5139,Y -104.4484,Z 184,A -126.4829,B 3.6647,C 0.3132,E1 3.5742,E2 219.4322} C_DIS
LIN {X -93.8437,Y -101.4672,Z 184,A -128.3024,B 3.665,C 0.3097,E1 3.5704,E2 221.2471} C_DIS
LIN {X -96.4567,Y -98.9867,Z 184,A -129.8358,B 3.6653,C 0.3071,E1 3.5673,E2 222.7856} C_DIS
LIN {X -99.2141,Y -96.2218,Z 184,A -131.5915,B 3.6654,C 0.3049,E1 3.5639,E2 224.5589} C_DIS
LIN {X -102.055,Y -93.2043,Z 184,A -133.2634,B 3.6658,C 0.3012,E1 3.5607,E2 226.2244} C_DIS
LIN {X -104.7085,Y -90.2119,Z 184,A -135.0311,B 3.666,C 0.2984,E1 3.5574,E2 228.0061} C_DIS
LIN {X -107.4961,Y -86.8716,Z 184,A -136.9218,B 3.6662,C 0.2951,E1 3.5541,E2 229.9077} C_DIS
LIN {X -110.0531,Y -83.6096,Z 184,A -138.598,B 3.6666,C 0.2912,E1 3.5512,E2 231.5779} C_DIS
LIN {X -112.1541,Y -80.7694,Z 184,A -140.1019,B 3.6668,C 0.2882,E1 3.5487,E2 233.0866} C_DIS
LIN {X -114.391,Y -77.5679,Z 184,A -141.8694,B 3.667,C 0.2853,E1 3.5459,E2 234.8729} C_DIS
LIN {X -116.6267,Y -74.165,Z 184,A -143.6143,B 3.6673,C 0.2818,E1 3.5432,E2 236.6246} C_DIS
LIN {X -118.9339,Y -70.4057,Z 184,A -145.4142,B 3.6676,C 0.2773,E1 3.5406,E2 238.4201} C_DIS
LIN {X -120.6987,Y -67.3356,Z 184,A -147.0602,B 3.6678,C 0.2747,E1 3.5383,E2 240.0886} C_DIS
LIN {X -122.7706,Y -63.4795,Z 184,A -148.8091,B 3.6682,C 0.2699,E1 3.5361,E2 241.8284} C_DIS
LIN {X -124.1245,Y -60.7847,Z 184,A -150.1019,B 3.6684,C 0.267,E1 3.5345,E2 243.1261} C_DIS
LIN {X -125.8097,Y -57.2204,Z 184,A -151.7953,B 3.6687,C 0.2632,E1 3.5325,E2 244.8264} C_DIS
LIN {X -127.2012,Y -54.0567,Z 184,A -153.2792,B 3.6689,C 0.2598,E1 3.5308,E2 246.3164} C_DIS
LIN {X -128.5069,Y -50.8747,Z 184,A -154.7567,B 3.6692,C 0.2564,E1 3.5293,E2 247.7998} C_DIS
LIN {X -129.548,Y -48.1557,Z 184,A -156.049,B 3.6693,C 0.2537,E1 3.528,E2 249.1024} C_DIS
LIN {X -130.8456,Y -44.5151,Z 184,A -157.6693,B 3.6696,C 0.2496,E1 3.5265,E2 250.7243} C_DIS
LIN {X -131.911,Y -41.2522,Z 184,A -159.145,B 3.6699,C 0.246,E1 3.5252,E2 252.2061} C_DIS
LIN {X -132.7751,Y -38.374,Z 184,A -160.4371,B 3.6701,C 0.2429,E1 3.5242,E2 253.5034} C_DIS
LIN {X -133.7566,Y -34.8054,Z 184,A -162.0295,B 3.6703,C 0.2391,E1 3.523,E2 255.1025} C_DIS
LIN {X -134.4107,Y -32.1772,Z 184,A -163.2234,B 3.6705,C 0.2364,E1 3.5223,E2 256.3048} C_DIS
LIN {X -135.1988,Y -28.6897,Z 184,A -164.7551,B 3.6707,C 0.2326,E1 3.5213,E2 257.8421} C_DIS
LIN {X -135.9035,Y -25.1493,Z 184,A -166.2872,B 3.671,C 0.2286,E1 3.5205,E2 259.3779} C_DIS
LIN {X -136.4498,Y -21.9917,Z 184,A -167.6612,B 3.6712,C 0.2252,E1 3.5199,E2 260.7569} C_DIS
LIN {X -136.8603,Y -19.2603,Z 184,A -168.8587,B 3.6714,C 0.2222,E1 3.5194,E2 261.9603} C_DIS
LIN {X -137.3302,Y -15.5781,Z 184,A -170.4544,B 3.6716,C 0.2182,E1 3.5189,E2 263.5624} C_DIS
LIN {X -137.6475,Y -12.464,Z 184,A -171.7957,B 3.6718,C 0.2148,E1 3.5185,E2 264.9085} C_DIS
LIN {X -137.8958,Y -9.3241,Z 184,A -173.1588,B 3.672,C 0.2114,E1 3.5182,E2 266.278} C_DIS
LIN {X -138.0713,Y -6.206,Z 184,A -174.4914,B 3.6722,C 0.2079,E1 3.518,E2 267.6145} C_DIS
LIN {X -138.2024,Y -1.5305,Z 184,A -176.5318,B 3.6725,C 0.203,E1 3.5179,E2 269.6665} C_DIS
LIN {X -138.2032,Y 1.4245,Z 184,A -177.8003,B 3.6727,C 0.1997,E1 3.5179,E2 270.9397} C_DIS
LIN {X -138.134,Y 4.6115,Z 184,A -179.1728,B 3.6729,C 0.1963,E1 3.518,E2 272.3177} C_DIS
LIN {X -137.9953,Y 7.7175,Z 184,A 179.4832,B 3.673,C 0.1929,E1 3.5182,E2 273.6679} C_DIS
LIN {X -137.6896,Y 11.9721,Z 184,A 177.6005,B 3.6733,C 0.1885,E1 3.5186,E2 275.5636} C_DIS
LIN {X -137.3302,Y 15.5781,Z 184,A 176.0727,B 3.6735,C 0.1844,E1 3.5191,E2 277.0937} C_DIS
LIN {X -136.9325,Y 18.7546,Z 184,A 174.6894,B 3.6736,C 0.181,E1 3.5196,E2 278.4831} C_DIS
LIN {X -136.2774,Y 23.025,Z 184,A 172.772,B 3.6739,C 0.1766,E1 3.5204,E2 280.415} C_DIS
LIN {X -135.6054,Y 26.7088,Z 184,A 171.2053,B 3.6741,C 0.1723,E1 3.5212,E2 281.9824} C_DIS
LIN {X -134.932,Y 29.9253,Z 184,A 169.7861,B 3.6742,C 0.1689,E1 3.5221,E2 283.4077} C_DIS
LIN {X -134.1829,Y 33.1225,Z 184,A 168.3784,B 3.6744,C 0.1654,E1 3.523,E2 284.8202} C_DIS
LIN {X -133.461,Y 35.914,Z 184,A 167.0792,B 3.6744,C 0.1626,E1 3.5239,E2 286.1314} C_DIS
LIN {X -132.404,Y 39.6415,Z 184,A 165.4527,B 3.6747,C 0.1584,E1 3.5252,E2 287.7593} C_DIS
LIN {X -131.4116,Y 42.8155,Z 184,A 164.0181,B 3.6748,C 0.1549,E1 3.5264,E2 289.1998} C_DIS
LIN {X -130.3049,Y 46.0747,Z 184,A 162.5345,B 3.675,C 0.1514,E1 3.5278,E2 290.6894} C_DIS
LIN {X -129.2799,Y 48.8714,Z 184,A 161.2201,B 3.675,C 0.1486,E1 3.5291,E2 292.0127} C_DIS
LIN {X -127.8831,Y 52.4222,Z 184,A 159.6075,B 3.6752,C 0.1446,E1 3.5307,E2 293.628} C_DIS
LIN {X -126.5358,Y 55.5957,Z 184,A 158.1234,B 3.6754,C 0.1412,E1 3.5324,E2 295.1178} C_DIS
LIN {X -125.1027,Y 58.7493,Z 184,A 156.6354,B 3.6755,C 0.1378,E1 3.5341,E2 296.6111} C_DIS
LIN {X -123.7504,Y 61.543,Z 184,A 155.2689,B 3.6756,C 0.1349,E1 3.5358,E2 297.9865} C_DIS
LIN {X -121.9809,Y 64.9833,Z 184,A 153.6346,B 3.6758,C 0.1311,E1 3.538,E2 299.6233} C_DIS
LIN {X -120.2686,Y 68.1009,Z 184,A 152.1073,B 3.6758,C 0.1278,E1 3.54,E2 301.1561} C_DIS
LIN {X -118.375,Y 71.3405,Z 184,A 150.3875,B 3.676,C 0.1249,E1 3.5425,E2 302.8949} C_DIS
LIN {X -116.1637,Y 74.8883,Z 184,A 148.7029,B 3.6761,C 0.1205,E1 3.545,E2 304.5721} C_DIS
LIN {X -114.2206,Y 77.8197,Z 184,A 147.1954,B 3.6762,C 0.1174,E1 3.5474,E2 306.0846} C_DIS
LIN {X -112.169,Y 80.7488,Z 184,A 145.6734,B 3.6763,C 0.1142,E1 3.5498,E2 307.6103} C_DIS
LIN {X -109.8446,Y 83.8822,Z 184,A 143.9045,B 3.6763,C 0.1114,E1 3.5528,E2 309.3966} C_DIS
LIN {X -107.3005,Y 87.1141,Z 184,A 142.2347,B 3.6765,C 0.1075,E1 3.5557,E2 311.0607} C_DIS
LIN {X -105.0143,Y 89.8568,Z 184,A 140.7114,B 3.6765,C 0.1046,E1 3.5585,E2 312.5881} C_DIS
LIN {X -102.6557,Y 92.5422,Z 184,A 139.1966,B 3.6767,C 0.1017,E1 3.5613,E2 314.1058} C_DIS
LIN {X -100.2443,Y 95.1489,Z 184,A 137.6654,B 3.6767,C 0.0991,E1 3.5643,E2 315.6431} C_DIS
LIN {X -97.7299,Y 97.7299,Z 184,A 136.1344,B 3.6768,C 0.0964,E1 3.5673,E2 317.1776} C_DIS
LIN {X -95.1675,Y 100.2268,Z 184,A 134.6082,B 3.6768,C 0.0938,E1 3.5703,E2 318.7079} C_DIS
LIN {X -92.5612,Y 102.6385,Z 184,A 133.1273,B 3.677,C 0.0911,E1 3.5734,E2 320.1888} C_DIS
LIN {X -89.8568,Y 105.0143,Z 184,A 131.5667,B 3.677,C 0.0888,E1 3.5767,E2 321.7566} C_DIS
LIN {X -87.1339,Y 107.2843,Z 184,A 130.061,B 3.677,C 0.0865,E1 3.58,E2 323.2656} C_DIS
LIN {X -84.317,Y 109.5121,Z 184,A 128.5393,B 3.6771,C 0.0842,E1 3.5833,E2 324.7903} C_DIS
LIN {X -81.4891,Y 111.6323,Z 184,A 127.0552,B 3.6771,C 0.0819,E1 3.5867,E2 326.2755} C_DIS
LIN {X -78.572,Y 113.7044,Z 184,A 125.5228,B 3.6772,C 0.0799,E1 3.5902,E2 327.8129} C_DIS
LIN {X -75.6515,Y 115.668,Z 184,A 124.0337,B 3.6772,C 0.0779,E1 3.5936,E2 329.3046} C_DIS
LIN {X -72.647,Y 117.5784,Z 184,A 122.4051,B 3.6772,C 0.0767,E1 3.5975,E2 330.9508} C_DIS
LIN {X -68.8859,Y 119.8206,Z 184,A 120.61,B 3.6773,C 0.0741,E1 3.6019,E2 332.7422} C_DIS
LIN {X -65.0497,Y 121.9458,Z 184,A 118.8288,B 3.6773,C 0.0715,E1 3.6062,E2 334.5175} C_DIS
LIN {X -61.9243,Y 123.5623,Z 184,A 117.3472,B 3.6774,C 0.0699,E1 3.6099,E2 336.0009} C_DIS
LIN {X -58.8395,Y 125.0604,Z 184,A 115.9084,B 3.6774,C 0.0684,E1 3.6135,E2 337.4409} C_DIS
LIN {X -55.641,Y 126.5161,Z 184,A 114.4266,B 3.6774,C 0.067,E1 3.6173,E2 338.9248} C_DIS
LIN {X -52.4678,Y 127.8647,Z 184,A 112.9783,B 3.6775,C 0.0657,E1 3.6211,E2 340.3745} C_DIS
LIN {X -49.2779,Y 129.1276,Z 184,A 111.5386,B 3.6775,C 0.0645,E1 3.6248,E2 341.8154} C_DIS
LIN {X -46.1206,Y 130.2884,Z 184,A 110.1369,B 3.6775,C 0.0633,E1 3.6285,E2 343.2171} C_DIS
LIN {X -43.2299,Y 131.2742,Z 184,A 108.8601,B 3.6775,C 0.0623,E1 3.6319,E2 344.4944} C_DIS
LIN {X -39.6415,Y 132.404,Z 184,A 107.2758,B 3.6775,C 0.0614,E1 3.6361,E2 346.0808} C_DIS
Enddeposition()
END
